            processes.reset.setActualStatus('Powering off the axis');
            // power off the axis
            processes.powerOff.start();
            processes.reset._state := 1;
        1:
            IF processes.powerOff.isIdle() THEN
                // regardless of whether power off worked or not, proceed    
                processes.reset._state := 2;
			END_IF
        2:
            // update the physical axis soft position limit values
            parts.physicalAxis.processes.writeParameter.start(parameterNumber := MC_AxisParameter.SWLimitNeg, value := config.minPositionLimitPhysicalAxis);
            processes.reset._state := 3;
        3:
            IF parts.physicalAxis.processes.writeParameter.isIdle() THEN
                IF parts.physicalAxis.processes.writeParameter.isGood() THEN
                    processes.reset._state := 4;
                ELSE
                    processes.reset.setActualStatus(CONCAT('Could not set the physical SWLimitNeg: ', parts.physicalAxis.processes.writeParameter.actualStatus));
                    processes.reset._state := 999;
				END_IF
			END_IF
        4:
            parts.physicalAxis.processes.writeParameter.start(parameterNumber := MC_AxisParameter.SWLimitPos, value := config.maxPositionLimitPhysicalAxis);
            processes.reset._state := 5;
        5:
            IF parts.physicalAxis.processes.writeParameter.isIdle() THEN
                IF parts.physicalAxis.processes.writeParameter.isGood() THEN
                    processes.reset._state := 6;
                ELSE
                    processes.reset.setActualStatus(CONCAT('Could not set the physical SWLimitPos: ', parts.physicalAxis.processes.writeParameter.actualStatus));
                    processes.reset._state := 999;
				END_IF
			END_IF
        6:
            parts.physicalAxis.processes.writeBoolParameter.start(parameterNumber := MC_AxisParameter.EnableLimitNeg, value := TRUE);
            processes.reset._state := 7;
        7:
            IF parts.physicalAxis.processes.writeBoolParameter.isIdle() THEN
                IF parts.physicalAxis.processes.writeBoolParameter.isGood() THEN
                    processes.reset._state := 8;
                ELSE
                    processes.reset.setActualStatus(CONCAT('Could not set the physical EnableLimitNeg: ', parts.physicalAxis.processes.writeBoolParameter.actualStatus));
                    processes.reset._state := 999;
				END_IF
			END_IF
        8:
            parts.physicalAxis.processes.writeBoolParameter.start(parameterNumber := MC_AxisParameter.EnableLimitPos, value := TRUE);
            processes.reset._state := 9;
        9:
            IF parts.physicalAxis.processes.writeBoolParameter.isIdle() THEN
                IF parts.physicalAxis.processes.writeBoolParameter.isGood() THEN
                    processes.reset._state := 10;
                ELSE
                    processes.reset.setActualStatus(CONCAT('Could not set the physical EnableLimitPos: ', parts.physicalAxis.processes.writeBoolParameter.actualStatus));
                    processes.reset._state := 999;
				END_IF
			END_IF
        10:
            // update the virtual axis soft position limit values
            parts.virtualAxis.processes.writeParameter.start(parameterNumber := MC_AxisParameter.SWLimitNeg, value := config.minPositionLimitVirtualAxis);
            processes.reset._state := 11;
        11:
            IF parts.virtualAxis.processes.writeParameter.isIdle() THEN
                IF parts.virtualAxis.processes.writeParameter.isGood() THEN
                    processes.reset._state := 12;
                ELSE
                    processes.reset.setActualStatus(CONCAT('Could not set the virtual SWLimitNeg: ', parts.virtualAxis.processes.writeParameter.actualStatus));
                    processes.reset._state := 999;
				END_IF
			END_IF
        12:
            parts.virtualAxis.processes.writeParameter.start(parameterNumber := MC_AxisParameter.SWLimitPos, value := config.maxPositionLimitVirtualAxis);
            processes.reset._state := 13;
        13:
            IF parts.virtualAxis.processes.writeParameter.isIdle() THEN
                IF parts.virtualAxis.processes.writeParameter.isGood() THEN
                    processes.reset._state := 14;
                ELSE
                    processes.reset.setActualStatus(CONCAT('Could not set the virtual SWLimitPos: ', parts.virtualAxis.processes.writeParameter.actualStatus));
                    processes.reset._state := 999;
				END_IF
			END_IF
        14:
            parts.virtualAxis.processes.writeBoolParameter.start(parameterNumber := MC_AxisParameter.EnableLimitNeg, value := TRUE);
            processes.reset._state := 15;
        15:
            IF parts.virtualAxis.processes.writeBoolParameter.isIdle() THEN
                IF parts.virtualAxis.processes.writeBoolParameter.isGood() THEN
                    processes.reset._state := 16;
                ELSE
                    processes.reset.setActualStatus(CONCAT('Could not set the virtual EnableLimitNeg: ', parts.virtualAxis.processes.writeBoolParameter.actualStatus));
                    processes.reset._state := 999;
				END_IF
			END_IF
        16:
            parts.virtualAxis.processes.writeBoolParameter.start(parameterNumber := MC_AxisParameter.EnableLimitPos, value := TRUE);
            processes.reset._state := 17;
        17:
            IF parts.virtualAxis.processes.writeBoolParameter.isIdle() THEN
                IF parts.virtualAxis.processes.writeBoolParameter.isGood() THEN
                    processes.reset._state := 18;
                ELSE
                    processes.reset.setActualStatus(CONCAT('Could not set the virtual EnableLimitPos: ', parts.virtualAxis.processes.writeBoolParameter.actualStatus));
                    processes.reset._state := 999;
				END_IF
			END_IF
            
        18:
            // reset the drive channel
            processes.reset.setActualStatus('Resetting the drive channel');
            driveChannel.processes.reset.start();
            processes.reset._state := 19;
        19:
            IF driveChannel.processes.reset.isIdle()  THEN
                IF driveChannel.processes.reset.isGood() THEN
                    processes.reset._state := 20;
                ELSE
                    processes.reset.setActualStatus('Could not reset the drive channels!');
                    processes.reset._state := 999;
                END_IF
            END_IF
            
        20:
            // try to acknowledge the safe state (if present)
            processes.reset.setActualStatus('Resetting safety');
            driveChannel.processes.acknowledgeSafetyError.start();
            processes.reset._state := 21;
        21:
            IF driveChannel.processes.acknowledgeSafetyError.isIdle()  THEN
                IF driveChannel.processes.acknowledgeSafetyError.isGood() THEN
                    processes.reset._state := 22;
                ELSE
                    processes.reset.setActualStatus('Cannot get out of safe state!');
                    processes.reset._state := 999;
                END_IF
            END_IF
        22:
            // reset the drive channel
            processes.reset.setActualStatus('Resetting the drive channel');
            driveChannel.processes.reset.start();
            processes.reset._state := 23;
        23:
            IF driveChannel.processes.reset.isIdle()  THEN
                IF driveChannel.processes.reset.isGood() THEN
                    processes.reset._state := 24;
                ELSE
                    processes.reset.setActualStatus('Could not reset the drive channels!');
                    processes.reset._state := 999;
                END_IF
            END_IF
        24:
            // update the drive channel
            processes.reset.setActualStatus('Updating the drive channel');
            driveChannel.processes.update.start();
            processes.reset._state := 25;
        25:
            IF driveChannel.processes.update.isIdle() AND driveChannel.processes.update.isIdle() THEN
                IF driveChannel.processes.update.isGood() AND driveChannel.processes.update.isGood() THEN
                    processes.reset._state := 26;
                ELSE
                    processes.reset.setActualStatus('Could not update the drive channel!');
                    processes.reset._state := 999;
                END_IF
            END_IF
        26:
            // reset the axis
            processes.reset.setActualStatus('Resetting the axes');
            parts.physicalAxis.processes.reset.start();
            parts.virtualAxis.processes.reset.start();
            processes.reset._state := 27;
        27:
            IF     parts.virtualAxis.processes.reset.isIdle() 
               AND parts.physicalAxis.processes.reset.isIdle()  THEN
                IF     parts.virtualAxis.processes.reset.isGood() 
                   AND parts.physicalAxis.processes.reset.isGood()  THEN
                    processes.reset._state := 1000;
                ELSE
                    processes.reset.setActualStatus('Could not reset the axes');
                    processes.reset._state := 999;
                END_IF
            END_IF
        999:
            // error!
            processes.reset.setBad();
            processes.reset.setFinished();
        1000:
            processes.reset.setActualStatus('Reset');
            // ok done
            processes.reset.setFinished();
            processes.reset.setGood();
    END_CASE
    
END_IF
END_METHOD

METHOD callOnce : BOOL
VAR_INPUT
    dcTime : LINT; 
	targetPosDeg  : LREAL; // degrees
	targetVeloDegPerSec : LREAL; // degrees/sec
	targetAccDegPerSec2  : LREAL; // degrees/sec2
    trackingStart : LREAL; // degrees
    modelDelta : LREAL; // degrees
END_VAR
VAR_IN_OUT
    isTracking : BOOL;
END_VAR
// run the setpoint generators
_setGen( 
    dcTime                      := dcTime,
    tracking                    := isTracking,
    virtual                     := parts.virtualAxis.axis_ref, 
    physical                    := parts.physicalAxis.axis_ref, 
    targetPos                   := targetPosDeg, 
    targetVelo                  := targetVeloDegPerSec, 
    targetAcc                   := targetAccDegPerSec2, 
    trackingStart               := trackingStart,
    velocityLimit               := config.velocityLimit,
    accelerationLimit           := config.accelerationLimit,
    minTrackingPositionSetpoint := config.minPositionSetpoint,
    maxTrackingPositionSetpoint := config.maxPositionSetpoint,
    minVirtualPositionSetpoint  := config.minPositionLimitVirtualAxis,
    maxVirtualPositionSetpoint  := config.maxPositionLimitVirtualAxis,
    limitReached                => setPosLimitReached);


// apply the position correction
IF parts.physicalAxis.axis_ref.Status.Homed THEN
    parts.physicalAxis.setPositionCorrection(lidaAveragePosition.degrees.value - parts.physicalAxis.axis_ref.NcToPlc.ActPosWithoutPosCorrection);
ELSE
    parts.physicalAxis.setPositionCorrection(0.0);
END_IF


// calculate the average and RMS deviation
_deviationCalculator(in := parts.physicalAxis.axis_ref.NcToPlc.ActPos - parts.physicalAxis.axis_ref.NcToPlc.SetPos );
deviation1SecAverage(newDegreesValue := _deviationCalculator.avg);
deviation1SecRMS(newDegreesValue := _deviationCalculator.rms);

// keep a local copy of the isTracking variable
_isTracking := isTracking;
END_METHOD

METHOD _moveAbsolute
VAR_INPUT
END_VAR
VAR
    positionDegrees : LREAL;
END_VAR
IF processes.moveAbsolute.isBusy() THEN
    
    IF NOT processes.moveAbsolute.isStarted() THEN
        
        targetStart(newDegreesValue := AxesMoveUnitsToDeg(units := processes.moveAbsolute.get.units, value := processes.moveAbsolute.get.value));
        
        parts.virtualAxis.processes.moveAbsolute.start(position := targetStart.degrees.value + processes.moveAbsolute.get.offset, maxVelocity := config.maxVelocitySetpoint);

        processes.moveAbsolute.setStarted();
            
	END_IF

    // update the statuses
    processes.moveAbsolute.statuses.busyStatus(isBusy := parts.virtualAxis.processes.moveAbsolute.statuses.busyStatus.isBusy);
    processes.moveAbsolute.statuses.healthStatus(
        isGood := parts.virtualAxis.processes.moveAbsolute.statuses.healthStatus.isGood,
        hasWarning := parts.virtualAxis.processes.moveAbsolute.statuses.healthStatus.hasWarning);
    processes.moveAbsolute.setActualStatus(parts.virtualAxis.processes.moveAbsolute.actualStatus);

END_IF
END_METHOD

METHOD _moveRelative
VAR_INPUT
END_VAR
VAR
    distanceDegrees : LREAL;
END_VAR
IF processes.moveRelative.isBusy() THEN
    
    IF NOT processes.moveRelative.isStarted() THEN
        
        distanceDegrees := AxesMoveUnitsToDeg(units := processes.moveRelative.get.units, value := processes.moveRelative.get.value);
        
        parts.virtualAxis.processes.moveRelative.start(distance := distanceDegrees, maxVelocity := config.maxVelocitySetpoint);
    
        processes.moveRelative.setStarted();
            
	END_IF

    // update the statuses
    processes.moveRelative.statuses.busyStatus(isBusy := parts.virtualAxis.processes.moveRelative.statuses.busyStatus.isBusy);
    processes.moveRelative.statuses.healthStatus(
        isGood := parts.virtualAxis.processes.moveRelative.statuses.healthStatus.isGood,
        hasWarning := parts.virtualAxis.processes.moveRelative.statuses.healthStatus.hasWarning);
    processes.moveRelative.setActualStatus(parts.virtualAxis.processes.moveRelative.actualStatus);

END_IF
END_METHOD

END_FUNCTION_BLOCK

// ---- MTCS/Axes/StateMachines/AxesRotationAxis.TcPOU
FUNCTION_BLOCK AxesRotationAxis EXTENDS SM_AxesRotationAxis
VAR_INPUT
END_VAR
VAR_OUTPUT
END_VAR
VAR 
    // setpoint generator
	{attribute 'OPC.UA.DA' := '0'}
    _setGen : AxesExternalSetpointGenerator;
    
    // helpers
	{attribute 'OPC.UA.DA' := '0'}
    _powerOnHelper : AxesPowerOnHelper;
	{attribute 'OPC.UA.DA' := '0'}
    _powerOffHelper : AxesPowerOffHelper;
	{attribute 'OPC.UA.DA' := '0'}
    _homingHelper : AxesHomingHelper;
	{attribute 'OPC.UA.DA' := '0'}
    _moveOutOfLimitSwitchHelper : AxesMoveOutOfLimitSwitchHelper;
	{attribute 'OPC.UA.DA' := '0'}
    _stopHelper : AxesStopHelper;
	{attribute 'OPC.UA.DA' := '0'}
    _quickStopHelper : AxesQuickStopHelper;
	{attribute 'OPC.UA.DA' := '0'}
    _setPositionHelper : AxesSetPositionHelper;
    
    // RMS and average setpoint deviation calculator
	{attribute 'OPC.UA.DA' := '0'}
    _deviationCalculator: AverageAndRmsCalculator;
    // local copy of the isTracking flag
	{attribute 'OPC.UA.DA' := '0'}
    _isTracking: BOOL;
	{attribute 'OPC.UA.DA' := '0'}
    _moveRelativeCalculator : AxesMoveRelativeCalculator;
	{attribute 'OPC.UA.DA' := '0'}
    _moveAbsoluteCalculator : AxesMoveAbsoluteCalculator;
    
END_VAR

_update();

_resetting();


_powerOnHelper(
    id                      := id,
    setpointGenerator       := _setGen,
    powerOn                 := processes.powerOn,
    stop                    := processes.stop,
    reset                   := processes.reset,
    virtual                 := parts.virtualAxis,
    physical                := parts.physicalAxis,
    targetStart             := targetStart,
    pAblAxis                := 0,
    pAblDriveChannel        := 0,
    pAblSetpointGenerator   := 0);
    
_powerOffHelper(
    setpointGenerator       := _setGen,
    powerOff                := processes.powerOff,
    stop                    := processes.stop,
    virtual                 := parts.virtualAxis,
    physical                := parts.physicalAxis,
    pAblAxis                := 0,
    pAblDriveChannel        := 0,
    pAblSetpointGenerator   := 0);


_moveOutOfLimitSwitchHelper(
    setpointGenerator               := _setGen,
    positiveLimitSwitchError        := positiveLimitSwitchError,
    negativeLimitSwitchError        := negativeLimitSwitchError,
    positiveLimitSwitchInput        := config.positiveLimitSwitchInput,
    negativeLimitSwitchInput        := config.negativeLimitSwitchInput,
    moveOutOfLimitSwitchDistance    := config.moveOutOfLimitSwitchDistance,
    moveOutOfLimitSwitch            := processes.moveOutOfLimitSwitch,
    moveRelative                    := processes.moveRelative,
    powerOn                         := processes.powerOn,
    reset                           := processes.reset,
    virtual                         := parts.virtualAxis,
    physical                        := parts.physicalAxis,
    driveChannel                    := mainDriveChannel);

_moveAbsolute();
_moveRelative();
_moveVelocity();

_stopHelper(
    setpointGenerator   := _setGen,
    stop                := processes.stop,
    virtual             := parts.virtualAxis,
    physical            := parts.physicalAxis);
    
_quickStopHelper(
    deceleration        := config.quickStopDeceleration, 
    jerk                := config.quickStopJerk,
    setpointGenerator   := _setGen,
    quickStop           := processes.quickStop,
    virtual             := parts.virtualAxis,
    physical            := parts.physicalAxis);
    
_setPositionHelper(
    setpointGenerator   := _setGen,
    setPosition         := processes.setPosition,
    virtual             := parts.virtualAxis,
    physical            := parts.physicalAxis);


_update();

METHOD callOnce : BOOL
VAR_INPUT
    dcTime : LINT; 
	targetPosDeg  : LREAL; // degrees
	targetVeloDegPerSec : LREAL; // degrees/sec
	targetAccDegPerSec2  : LREAL; // degrees/sec2
    trackingStart : LREAL; // degrees
END_VAR
VAR_IN_OUT
    isTracking : BOOL;
END_VAR
// run the setpoint generators
_setGen( 
    dcTime                      := dcTime,
    tracking                    := isTracking,
    virtual                     := parts.virtualAxis.axis_ref, 
    physical                    := parts.physicalAxis.axis_ref, 
    targetPos                   := targetPosDeg, 
    targetVelo                  := targetVeloDegPerSec, 
    targetAcc                   := targetAccDegPerSec2, 
    trackingStart               := trackingStart,
    velocityLimit               := config.velocityLimit,
    accelerationLimit           := config.accelerationLimit,
    minTrackingPositionSetpoint := config.minPositionSetpoint,
    maxTrackingPositionSetpoint := config.maxPositionSetpoint,
    minVirtualPositionSetpoint  := config.minPositionLimitVirtualAxis,
    maxVirtualPositionSetpoint  := config.maxPositionLimitVirtualAxis,
    limitReached                => setPosLimitReached);

// calculate the average and RMS deviation
_deviationCalculator(in := parts.physicalAxis.axis_ref.NcToPlc.ActPos - parts.physicalAxis.axis_ref.NcToPlc.SetPos );
deviation1SecAverage(newDegreesValue := _deviationCalculator.avg);
deviation1SecRMS(newDegreesValue := _deviationCalculator.rms);

// keep a local copy of the isTracking variable
_isTracking := isTracking;
END_METHOD

METHOD _moveVelocity
VAR_INPUT
END_VAR
VAR
    velocityDegPerSec : LREAL;
END_VAR
IF processes.moveVelocity.isBusy() THEN
    
    IF NOT processes.moveVelocity.isStarted() THEN
        
        velocityDegPerSec := AxesMoveVelocityUnitsToDegPerSec(units := processes.moveVelocity.get.units, value := processes.moveVelocity.get.value);
        
        parts.virtualAxis.processes.moveVelocity.start(value := velocityDegPerSec);
    
        processes.moveVelocity.setStarted();
            
	END_IF

    // update the statuses
    processes.moveVelocity.statuses.busyStatus(isBusy := parts.virtualAxis.processes.moveVelocity.statuses.busyStatus.isBusy);
    processes.moveVelocity.statuses.healthStatus(
        isGood := parts.virtualAxis.processes.moveVelocity.statuses.healthStatus.isGood,
        hasWarning := parts.virtualAxis.processes.moveVelocity.statuses.healthStatus.hasWarning);
    processes.moveVelocity.setActualStatus(parts.virtualAxis.processes.moveVelocity.actualStatus);

END_IF
END_METHOD

METHOD _update : LREAL
VAR_INPUT
END_VAR
VAR
END_VAR
// update the superclass
SUPER^(
    config := config,
    driveChannel := driveChannel,
    mainDriveChannel := mainDriveChannel);
    
// update the limit switches
positiveLimitSwitchError := NOT GETBIT32(inVal32 := INT_TO_DWORD(driveChannel.digitalInputs), bitNo := config.positiveLimitSwitchInput);
negativeLimitSwitchError := NOT GETBIT32(inVal32 := INT_TO_DWORD(driveChannel.digitalInputs), bitNo := config.negativeLimitSwitchInput);

// update the actual position/velocity/acceleration
actPos(newDegreesValue := parts.physicalAxis.axis_ref.NcToPlc.ActPos);
actVelo(newDegreesPerSecondValue := parts.physicalAxis.axis_ref.NcToPlc.ActVelo);
actAcc(newDegreesPerSquareSecondValue := parts.physicalAxis.axis_ref.NcToPlc.ActAcc);
setPos(newDegreesValue := parts.physicalAxis.axis_ref.NcToPlc.SetPos);
setVelo(newDegreesPerSecondValue := parts.physicalAxis.axis_ref.NcToPlc.SetVelo);
setAcc(newDegreesPerSquareSecondValue := parts.physicalAxis.axis_ref.NcToPlc.SetAcc);
IF parts.physicalAxis.axis_ref.Status.ExtSetPointGenEnabled THEN
    targetPos(newDegreesValue := parts.physicalAxis.axis_ref.PlcToNc.ExtSetPos);
    targetOffset(newDegreesValue := parts.virtualAxis.actPos.degrees.value - targetStart.degrees.value);
ELSE
    targetPos(newDegreesValue := parts.physicalAxis.axis_ref.NcToPlc.TargetPos);
    targetOffset(newDegreesValue := 0.0);
END_IF

// update the actual torque feedback on the telescope side
actTorque(newNewtonmeterValue := driveChannel.actualTorqueFeedback.newtonmeter.value * 1440);
END_METHOD

METHOD _moveRelative
VAR_INPUT
END_VAR
VAR
    distanceDegrees : LREAL;
END_VAR
IF processes.moveRelative.isBusy() THEN
    
    IF NOT processes.moveRelative.isStarted() THEN
        
        distanceDegrees := AxesMoveUnitsToDeg(units := processes.moveRelative.get.units, value := processes.moveRelative.get.value);
        
        parts.virtualAxis.processes.moveRelative.start(distance := distanceDegrees, maxVelocity := config.maxVelocitySetpoint);
    
        processes.moveRelative.setStarted();
    ELSE
        
        // update the statuses
        processes.moveRelative.statuses.healthStatus(
            isGood := parts.virtualAxis.processes.moveRelative.statuses.healthStatus.isGood,
            hasWarning := parts.virtualAxis.processes.moveRelative.statuses.healthStatus.hasWarning);
        processes.moveRelative.setActualStatus(parts.virtualAxis.processes.moveRelative.actualStatus);
        processes.moveRelative.statuses.busyStatus(isBusy := parts.virtualAxis.processes.moveRelative.statuses.busyStatus.isBusy);
    
	END_IF
END_IF
(*IF processes.moveRelative.isBusy() THEN
    
    IF NOT processes.moveRelative.isStarted() THEN
        
        distanceDegrees := AxesMoveUnitsToDeg(units := processes.moveRelative.get.units, value := processes.moveRelative.get.value);
        
        _moveRelativeCalculator(
            distance     := distanceDegrees, 
            trackingVelo := _setGen.targetVelo,
            minPos       := config.minPositionLimitVirtualAxis,
            maxPos       := config.maxPositionLimitVirtualAxis,
            actPos       := actPos.degrees.value,
            doMostTravel := processes.moveRelative.get.preferMostTravel);
        
        IF _moveRelativeCalculator.outOfRange THEN
            processes.moveRelative.setFinished();
            processes.moveRelative.setActualStatus('Out of limits!');
            processes.moveRelative.setBad();
        ELSE
            parts.virtualAxis.processes.moveRelative.start(distance := _moveRelativeCalculator.adjustedDistance, maxVelocity := config.maxVelocitySetpoint);
            processes.moveRelative.setStarted();
        END_IF
        
    ELSE
        // update the statuses
        processes.moveRelative.statuses.busyStatus(isBusy := parts.virtualAxis.processes.moveRelative.statuses.busyStatus.isBusy);
        processes.moveRelative.statuses.healthStatus(
            isGood := parts.virtualAxis.processes.moveRelative.statuses.healthStatus.isGood,
            hasWarning := parts.virtualAxis.processes.moveRelative.statuses.healthStatus.hasWarning);
        processes.moveRelative.setActualStatus(parts.virtualAxis.processes.moveRelative.actualStatus);

	END_IF

END_IF*)
END_METHOD

METHOD _moveAbsolute
VAR_INPUT
END_VAR
VAR
    positionDegrees : LREAL;
END_VAR
IF processes.moveAbsolute.isBusy() THEN
    
    IF NOT processes.moveAbsolute.isStarted() THEN
        
        targetStart(newDegreesValue := AxesMoveUnitsToDeg(units := processes.moveAbsolute.get.units, value := processes.moveAbsolute.get.value));
        
        parts.virtualAxis.processes.moveAbsolute.start(position := targetStart.degrees.value + processes.moveAbsolute.get.offset, maxVelocity := config.maxVelocitySetpoint);

        processes.moveAbsolute.setStarted();
        
    END_IF

    IF parts.virtualAxis.processes.moveAbsolute.isIdle() THEN
        
        IF parts.virtualAxis.processes.moveAbsolute.isGood() THEN
            processes.moveAbsolute.setGood();
        ELSE
            processes.moveAbsolute.setBad();
		END_IF
        
        processes.moveAbsolute.setActualStatus(parts.virtualAxis.processes.moveAbsolute.actualStatus);
        processes.moveAbsolute.setFinished();
    
	END_IF
    
END_IF
(*IF processes.moveAbsolute.isBusy() THEN
    
    IF NOT processes.moveAbsolute.isStarted() THEN
        
        _moveAbsoluteCalculator(
            targetPos := AxesMoveUnitsToDeg(units := processes.moveAbsolute.get.units, value := processes.moveAbsolute.get.value),
            trackingVelo := _setGen.targetVelo,
            minPos := config.minPositionLimitVirtualAxis,
            maxPos := config.maxPositionLimitVirtualAxis,
            actPos := parts.virtualAxis.actPos.degrees.value,
            doMostTravel := FALSE); // get there the quickest possible
        
        IF _moveAbsoluteCalculator.outOfRange THEN
            processes.moveAbsolute.setActualStatus('Out of limits!');
            processes.moveAbsolute.setBad();
            processes.moveAbsolute.setFinished();
        ELSE
            targetStart(newDegreesValue := _moveAbsoluteCalculator.adjustedPos);
            parts.virtualAxis.processes.moveAbsolute.start(position := targetStart.degrees.value, maxVelocity := config.maxVelocitySetpoint);
            processes.moveAbsolute.setStarted();
		END_IF
            
    ELSE
        // update the statuses
        processes.moveAbsolute.statuses.busyStatus(isBusy := parts.virtualAxis.processes.moveAbsolute.statuses.busyStatus.isBusy);
        processes.moveAbsolute.statuses.healthStatus(
            isGood := parts.virtualAxis.processes.moveAbsolute.statuses.healthStatus.isGood,
            hasWarning := parts.virtualAxis.processes.moveAbsolute.statuses.healthStatus.hasWarning);
        processes.moveAbsolute.setActualStatus(parts.virtualAxis.processes.moveAbsolute.actualStatus);

	END_IF

END_IF*)
END_METHOD

METHOD _resetting : LREAL
VAR_INPUT
END_VAR
IF processes.reset.isBusy() THEN
    
    IF NOT processes.reset.isStarted() THEN
        processes.reset._state := 0;
        processes.reset.setStarted();
	END_IF
    
    CASE processes.reset._state OF
        0:
            // reset all processes so that they are green again
            processes.moveAbsolute.resetIfIdle();
            processes.moveOutOfLimitSwitch.resetIfIdle();
            processes.moveRelative.resetIfIdle();
            processes.moveVelocity.resetIfIdle();
            processes.powerOff.resetIfIdle();
            processes.powerOn.resetIfIdle();
            processes.quickStop.resetIfIdle();
            processes.setPosition.resetIfIdle();
            processes.stop.resetIfIdle();
            
            processes.reset.setActualStatus('Powering off the axis');
            // power off the axis
            processes.powerOff.start();
            processes.reset._state := 1;
        1:
            IF processes.powerOff.isIdle() THEN
                // regardless of whether power off worked or not, proceed    
                processes.reset._state := 2;
			END_IF
        2:
            // update the physical axis soft position limit values
            parts.physicalAxis.processes.writeParameter.start(parameterNumber := MC_AxisParameter.AxisEncoderOffset, value := config.motorEncoderOffset);
            processes.reset._state := 3;
        3:
            IF parts.physicalAxis.processes.writeParameter.isIdle() THEN
                IF parts.physicalAxis.processes.writeParameter.isGood() THEN
                    processes.reset._state := 4;
                ELSE
                    processes.reset.setActualStatus(CONCAT('Could not set the motor encoder offset: ', parts.physicalAxis.processes.writeParameter.actualStatus));
                    processes.reset._state := 999;
				END_IF
			END_IF
        4:
            // update the physical axis soft position limit values
            parts.physicalAxis.processes.writeParameter.start(parameterNumber := MC_AxisParameter.SWLimitNeg, value := config.minPositionLimitPhysicalAxis);
            processes.reset._state := 5;
        5:
            IF parts.physicalAxis.processes.writeParameter.isIdle() THEN
                IF parts.physicalAxis.processes.writeParameter.isGood() THEN
                    processes.reset._state := 6;
                ELSE
                    processes.reset.setActualStatus(CONCAT('Could not set the physical SWLimitNeg: ', parts.physicalAxis.processes.writeParameter.actualStatus));
                    processes.reset._state := 999;
				END_IF
			END_IF
        6:
            parts.physicalAxis.processes.writeParameter.start(parameterNumber := MC_AxisParameter.SWLimitPos, value := config.maxPositionLimitPhysicalAxis);
            processes.reset._state := 7;
        7:
            IF parts.physicalAxis.processes.writeParameter.isIdle() THEN
                IF parts.physicalAxis.processes.writeParameter.isGood() THEN
                    processes.reset._state := 8;
                ELSE
                    processes.reset.setActualStatus(CONCAT('Could not set the physical SWLimitPos: ', parts.physicalAxis.processes.writeParameter.actualStatus));
                    processes.reset._state := 999;
				END_IF
			END_IF
        8:
            parts.physicalAxis.processes.writeBoolParameter.start(parameterNumber := MC_AxisParameter.EnableLimitNeg, value := TRUE);
            processes.reset._state := 9;
        9:
            IF parts.physicalAxis.processes.writeBoolParameter.isIdle() THEN
                IF parts.physicalAxis.processes.writeBoolParameter.isGood() THEN
                    processes.reset._state := 10;
                ELSE
                    processes.reset.setActualStatus(CONCAT('Could not set the physical EnableLimitNeg: ', parts.physicalAxis.processes.writeBoolParameter.actualStatus));
                    processes.reset._state := 999;
				END_IF
			END_IF
        10:
            parts.physicalAxis.processes.writeBoolParameter.start(parameterNumber := MC_AxisParameter.EnableLimitPos, value := TRUE);
            processes.reset._state := 11;
        11:
            IF parts.physicalAxis.processes.writeBoolParameter.isIdle() THEN
                IF parts.physicalAxis.processes.writeBoolParameter.isGood() THEN
                    processes.reset._state := 12;
                ELSE
                    processes.reset.setActualStatus(CONCAT('Could not set the physical EnableLimitPos: ', parts.physicalAxis.processes.writeBoolParameter.actualStatus));
                    processes.reset._state := 999;
				END_IF
			END_IF
        12:
            // update the virtual axis soft position limit values
            parts.virtualAxis.processes.writeParameter.start(parameterNumber := MC_AxisParameter.SWLimitNeg, value := config.minPositionLimitVirtualAxis);
            processes.reset._state := 13;
        13:
            IF parts.virtualAxis.processes.writeParameter.isIdle() THEN
                IF parts.virtualAxis.processes.writeParameter.isGood() THEN
                    processes.reset._state := 14;
                ELSE
                    processes.reset.setActualStatus(CONCAT('Could not set the virtual SWLimitNeg: ', parts.virtualAxis.processes.writeParameter.actualStatus));
                    processes.reset._state := 999;
				END_IF
			END_IF
        14:
            parts.virtualAxis.processes.writeParameter.start(parameterNumber := MC_AxisParameter.SWLimitPos, value := config.maxPositionLimitVirtualAxis);
            processes.reset._state := 15;
        15:
            IF parts.virtualAxis.processes.writeParameter.isIdle() THEN
                IF parts.virtualAxis.processes.writeParameter.isGood() THEN
                    processes.reset._state := 16;
                ELSE
                    processes.reset.setActualStatus(CONCAT('Could not set the virtual SWLimitPos: ', parts.virtualAxis.processes.writeParameter.actualStatus));
                    processes.reset._state := 999;
				END_IF
			END_IF
        16:
            parts.virtualAxis.processes.writeBoolParameter.start(parameterNumber := MC_AxisParameter.EnableLimitNeg, value := TRUE);
            processes.reset._state := 17;
        17:
            IF parts.virtualAxis.processes.writeBoolParameter.isIdle() THEN
                IF parts.virtualAxis.processes.writeBoolParameter.isGood() THEN
                    processes.reset._state := 18;
                ELSE
                    processes.reset.setActualStatus(CONCAT('Could not set the virtual EnableLimitNeg: ', parts.virtualAxis.processes.writeBoolParameter.actualStatus));
                    processes.reset._state := 999;
				END_IF
			END_IF
        18:
            parts.virtualAxis.processes.writeBoolParameter.start(parameterNumber := MC_AxisParameter.EnableLimitPos, value := TRUE);
            processes.reset._state := 19;
        19:
            IF parts.virtualAxis.processes.writeBoolParameter.isIdle() THEN
                IF parts.virtualAxis.processes.writeBoolParameter.isGood() THEN
                    processes.reset._state := 20;
                ELSE
                    processes.reset.setActualStatus(CONCAT('Could not set the virtual EnableLimitPos: ', parts.virtualAxis.processes.writeBoolParameter.actualStatus));
                    processes.reset._state := 999;
				END_IF
			END_IF
            
        20:
            // try to acknowledge the safe state (if present)
            processes.reset.setActualStatus('Resetting safety');
            driveChannel.processes.acknowledgeSafetyError.start();
            processes.reset._state := 21;
        21:
            IF driveChannel.processes.acknowledgeSafetyError.isIdle()  THEN
                IF driveChannel.processes.acknowledgeSafetyError.isGood() THEN
                    processes.reset._state := 22;
                ELSE
                    processes.reset.setActualStatus('Cannot get out of safe state!');
                    processes.reset._state := 999;
                END_IF
            END_IF
        22:
            // reset the drive channel
            processes.reset.setActualStatus('Resetting the drive channel');
            driveChannel.processes.reset.start();
            processes.reset._state := 23;
        23:
            IF driveChannel.processes.reset.isIdle()  THEN
                IF driveChannel.processes.reset.isGood() THEN
                    processes.reset._state := 24;
                ELSE
                    processes.reset.setActualStatus('Could not reset the drive channels!');
                    processes.reset._state := 999;
                END_IF
            END_IF
        24:
            // update the drive channel
            processes.reset.setActualStatus('Updating the drive channel');
            driveChannel.processes.update.start();
            processes.reset._state := 25;
        25:
            IF driveChannel.processes.update.isIdle() AND driveChannel.processes.update.isIdle() THEN
                IF driveChannel.processes.update.isGood() AND driveChannel.processes.update.isGood() THEN
                    processes.reset._state := 26;
                ELSE
                    processes.reset.setActualStatus('Could not update the drive channel!');
                    processes.reset._state := 999;
                END_IF
            END_IF
        26:
            // reset the axis
            processes.reset.setActualStatus('Resetting the axes');
            parts.physicalAxis.processes.reset.start();
            parts.virtualAxis.processes.reset.start();
            processes.reset._state := 27;
        27:
            IF     parts.virtualAxis.processes.reset.isIdle() 
               AND parts.physicalAxis.processes.reset.isIdle()  THEN
                IF     parts.virtualAxis.processes.reset.isGood() 
                   AND parts.physicalAxis.processes.reset.isGood()  THEN
                    processes.reset._state := 1000;
                ELSE
                    processes.reset.setActualStatus('Could not reset the axes');
                    processes.reset._state := 999;
                END_IF
            END_IF
        999:
            // error!
            processes.reset.setBad();
            processes.reset.setFinished();
        1000:
            processes.reset.setActualStatus('Reset');
            // ok done
            processes.reset.setFinished();
            processes.reset.setGood();
    END_CASE
    
END_IF
END_METHOD

END_FUNCTION_BLOCK

// ---- MTCS/Axes/StateMachines/AxesIO.TcPOU
FUNCTION_BLOCK AxesIO EXTENDS SM_AxesIO
VAR_INPUT
END_VAR
VAR_OUTPUT
END_VAR
VAR
    _testVar : BOOL; // without any variable, the superclass attributes are not visible in the UA address space
END_VAR

SUPER^();

// do stuff

//SUPER^();

END_FUNCTION_BLOCK

// ---- MTCS/Axes/StateMachines/AxesPointingModelsSetup.TcPOU
FUNCTION_BLOCK AxesPointingModelsSetup EXTENDS SM_AxesPointingModelsSetup
VAR_INPUT
END_VAR
VAR_OUTPUT
END_VAR
VAR
	{attribute 'OPC.UA.DA' := '0'}
    _onFirstStartCurrentAction : INT;
END_VAR

SUPER^();

_onFirstStart();

METHOD FB_init : BOOL
VAR_INPUT
	bInitRetains : BOOL; // if TRUE, the retain variables are initialized (warm start / cold start)
	bInCopyCode : BOOL;  // if TRUE, the instance afterwards gets moved into the copy code (online change)
END_VAR
parts.model0.parts.configManager.configure(
    editableConfigAddress       := ADR(parts.model0.editableConfig),
    activeConfigAddress         := ADR(parts.model0.config),
    configLength                := SIZEOF(parts.model0.editableConfig),
    editableConfigSymbolName    := CONCAT(CONCAT(GLOBAL.config.AXES_TPOINT_EDITABLE_CONFIG_SYMBOL_PREFIX, 'model0'), GLOBAL.config.AXES_TPOINT_EDITABLE_CONFIG_SYMBOL_SUFFIX),
    activeConfigSymbolName      := CONCAT(CONCAT(GLOBAL.config.AXES_TPOINT_ACTIVE_CONFIG_SYMBOL_PREFIX, 'model0'), GLOBAL.config.AXES_TPOINT_ACTIVE_CONFIG_SYMBOL_SUFFIX),
    configFilePath              := CONCAT(CONCAT(GLOBAL.config.AXES_TPOINT_CONFIG_FILE_PATH_PREFIX, 'model0'), GLOBAL.config.AXES_TPOINT_CONFIG_FILE_PATH_SUFFIX));
    
parts.model1.parts.configManager.configure(
    editableConfigAddress       := ADR(parts.model1.editableConfig),
    activeConfigAddress         := ADR(parts.model1.config),
    configLength                := SIZEOF(parts.model1.editableConfig),
    editableConfigSymbolName    := CONCAT(CONCAT(GLOBAL.config.AXES_TPOINT_EDITABLE_CONFIG_SYMBOL_PREFIX, 'model1'), GLOBAL.config.AXES_TPOINT_EDITABLE_CONFIG_SYMBOL_SUFFIX),
    activeConfigSymbolName      := CONCAT(CONCAT(GLOBAL.config.AXES_TPOINT_ACTIVE_CONFIG_SYMBOL_PREFIX, 'model1'), GLOBAL.config.AXES_TPOINT_ACTIVE_CONFIG_SYMBOL_SUFFIX),
    configFilePath              := CONCAT(CONCAT(GLOBAL.config.AXES_TPOINT_CONFIG_FILE_PATH_PREFIX, 'model1'), GLOBAL.config.AXES_TPOINT_CONFIG_FILE_PATH_SUFFIX));
    
parts.model2.parts.configManager.configure(
    editableConfigAddress       := ADR(parts.model2.editableConfig),
    activeConfigAddress         := ADR(parts.model2.config),
    configLength                := SIZEOF(parts.model2.editableConfig),
    editableConfigSymbolName    := CONCAT(CONCAT(GLOBAL.config.AXES_TPOINT_EDITABLE_CONFIG_SYMBOL_PREFIX, 'model2'), GLOBAL.config.AXES_TPOINT_EDITABLE_CONFIG_SYMBOL_SUFFIX),
    activeConfigSymbolName      := CONCAT(CONCAT(GLOBAL.config.AXES_TPOINT_ACTIVE_CONFIG_SYMBOL_PREFIX, 'model2'), GLOBAL.config.AXES_TPOINT_ACTIVE_CONFIG_SYMBOL_SUFFIX),
    configFilePath              := CONCAT(CONCAT(GLOBAL.config.AXES_TPOINT_CONFIG_FILE_PATH_PREFIX, 'model2'), GLOBAL.config.AXES_TPOINT_CONFIG_FILE_PATH_SUFFIX));
parts.model3.parts.configManager.configure(
    editableConfigAddress       := ADR(parts.model3.editableConfig),
    activeConfigAddress         := ADR(parts.model3.config),
    configLength                := SIZEOF(parts.model3.editableConfig),
    editableConfigSymbolName    := CONCAT(CONCAT(GLOBAL.config.AXES_TPOINT_EDITABLE_CONFIG_SYMBOL_PREFIX, 'model3'), GLOBAL.config.AXES_TPOINT_EDITABLE_CONFIG_SYMBOL_SUFFIX),
    activeConfigSymbolName      := CONCAT(CONCAT(GLOBAL.config.AXES_TPOINT_ACTIVE_CONFIG_SYMBOL_PREFIX, 'model3'), GLOBAL.config.AXES_TPOINT_ACTIVE_CONFIG_SYMBOL_SUFFIX),
    configFilePath              := CONCAT(CONCAT(GLOBAL.config.AXES_TPOINT_CONFIG_FILE_PATH_PREFIX, 'model3'), GLOBAL.config.AXES_TPOINT_CONFIG_FILE_PATH_SUFFIX));
parts.model4.parts.configManager.configure(
    editableConfigAddress       := ADR(parts.model4.editableConfig),
    activeConfigAddress         := ADR(parts.model4.config),
    configLength                := SIZEOF(parts.model4.editableConfig),
    editableConfigSymbolName    := CONCAT(CONCAT(GLOBAL.config.AXES_TPOINT_EDITABLE_CONFIG_SYMBOL_PREFIX, 'model4'), GLOBAL.config.AXES_TPOINT_EDITABLE_CONFIG_SYMBOL_SUFFIX),
    activeConfigSymbolName      := CONCAT(CONCAT(GLOBAL.config.AXES_TPOINT_ACTIVE_CONFIG_SYMBOL_PREFIX, 'model4'), GLOBAL.config.AXES_TPOINT_ACTIVE_CONFIG_SYMBOL_SUFFIX),
    configFilePath              := CONCAT(CONCAT(GLOBAL.config.AXES_TPOINT_CONFIG_FILE_PATH_PREFIX, 'model4'), GLOBAL.config.AXES_TPOINT_CONFIG_FILE_PATH_SUFFIX));
parts.model5.parts.configManager.configure(
    editableConfigAddress       := ADR(parts.model5.editableConfig),
    activeConfigAddress         := ADR(parts.model5.config),
    configLength                := SIZEOF(parts.model5.editableConfig),
    editableConfigSymbolName    := CONCAT(CONCAT(GLOBAL.config.AXES_TPOINT_EDITABLE_CONFIG_SYMBOL_PREFIX, 'model5'), GLOBAL.config.AXES_TPOINT_EDITABLE_CONFIG_SYMBOL_SUFFIX),
    activeConfigSymbolName      := CONCAT(CONCAT(GLOBAL.config.AXES_TPOINT_ACTIVE_CONFIG_SYMBOL_PREFIX, 'model5'), GLOBAL.config.AXES_TPOINT_ACTIVE_CONFIG_SYMBOL_SUFFIX),
    configFilePath              := CONCAT(CONCAT(GLOBAL.config.AXES_TPOINT_CONFIG_FILE_PATH_PREFIX, 'model5'), GLOBAL.config.AXES_TPOINT_CONFIG_FILE_PATH_SUFFIX));
parts.model6.parts.configManager.configure(
    editableConfigAddress       := ADR(parts.model6.editableConfig),
    activeConfigAddress         := ADR(parts.model6.config),
    configLength                := SIZEOF(parts.model6.editableConfig),
    editableConfigSymbolName    := CONCAT(CONCAT(GLOBAL.config.AXES_TPOINT_EDITABLE_CONFIG_SYMBOL_PREFIX, 'model6'), GLOBAL.config.AXES_TPOINT_EDITABLE_CONFIG_SYMBOL_SUFFIX),
    activeConfigSymbolName      := CONCAT(CONCAT(GLOBAL.config.AXES_TPOINT_ACTIVE_CONFIG_SYMBOL_PREFIX, 'model6'), GLOBAL.config.AXES_TPOINT_ACTIVE_CONFIG_SYMBOL_SUFFIX),
    configFilePath              := CONCAT(CONCAT(GLOBAL.config.AXES_TPOINT_CONFIG_FILE_PATH_PREFIX, 'model6'), GLOBAL.config.AXES_TPOINT_CONFIG_FILE_PATH_SUFFIX));
parts.model7.parts.configManager.configure(
    editableConfigAddress       := ADR(parts.model7.editableConfig),
    activeConfigAddress         := ADR(parts.model7.config),
    configLength                := SIZEOF(parts.model7.editableConfig),
    editableConfigSymbolName    := CONCAT(CONCAT(GLOBAL.config.AXES_TPOINT_EDITABLE_CONFIG_SYMBOL_PREFIX, 'model7'), GLOBAL.config.AXES_TPOINT_EDITABLE_CONFIG_SYMBOL_SUFFIX),
    activeConfigSymbolName      := CONCAT(CONCAT(GLOBAL.config.AXES_TPOINT_ACTIVE_CONFIG_SYMBOL_PREFIX, 'model7'), GLOBAL.config.AXES_TPOINT_ACTIVE_CONFIG_SYMBOL_SUFFIX),
    configFilePath              := CONCAT(CONCAT(GLOBAL.config.AXES_TPOINT_CONFIG_FILE_PATH_PREFIX, 'model7'), GLOBAL.config.AXES_TPOINT_CONFIG_FILE_PATH_SUFFIX));
parts.model8.parts.configManager.configure(
    editableConfigAddress       := ADR(parts.model8.editableConfig),
    activeConfigAddress         := ADR(parts.model8.config),
    configLength                := SIZEOF(parts.model8.editableConfig),
    editableConfigSymbolName    := CONCAT(CONCAT(GLOBAL.config.AXES_TPOINT_EDITABLE_CONFIG_SYMBOL_PREFIX, 'model8'), GLOBAL.config.AXES_TPOINT_EDITABLE_CONFIG_SYMBOL_SUFFIX),
    activeConfigSymbolName      := CONCAT(CONCAT(GLOBAL.config.AXES_TPOINT_ACTIVE_CONFIG_SYMBOL_PREFIX, 'model8'), GLOBAL.config.AXES_TPOINT_ACTIVE_CONFIG_SYMBOL_SUFFIX),
    configFilePath              := CONCAT(CONCAT(GLOBAL.config.AXES_TPOINT_CONFIG_FILE_PATH_PREFIX, 'model8'), GLOBAL.config.AXES_TPOINT_CONFIG_FILE_PATH_SUFFIX));
parts.model9.parts.configManager.configure(
    editableConfigAddress       := ADR(parts.model9.editableConfig),
    activeConfigAddress         := ADR(parts.model9.config),
    configLength                := SIZEOF(parts.model9.editableConfig),
    editableConfigSymbolName    := CONCAT(CONCAT(GLOBAL.config.AXES_TPOINT_EDITABLE_CONFIG_SYMBOL_PREFIX, 'model9'), GLOBAL.config.AXES_TPOINT_EDITABLE_CONFIG_SYMBOL_SUFFIX),
    activeConfigSymbolName      := CONCAT(CONCAT(GLOBAL.config.AXES_TPOINT_ACTIVE_CONFIG_SYMBOL_PREFIX, 'model9'), GLOBAL.config.AXES_TPOINT_ACTIVE_CONFIG_SYMBOL_SUFFIX),
    configFilePath              := CONCAT(CONCAT(GLOBAL.config.AXES_TPOINT_CONFIG_FILE_PATH_PREFIX, 'model9'), GLOBAL.config.AXES_TPOINT_CONFIG_FILE_PATH_SUFFIX));
END_METHOD

METHOD _onFirstStart
VAR_INPUT
END_VAR
CASE _onFirstStartCurrentAction OF
    0:
        // start loading the config from XML file
        parts.model0.parts.configManager.processes.load.start(parts.model0.parts.configManager.processes.load.set.filePath);
        parts.model1.parts.configManager.processes.load.start(parts.model1.parts.configManager.processes.load.set.filePath);
        parts.model2.parts.configManager.processes.load.start(parts.model2.parts.configManager.processes.load.set.filePath);
        parts.model3.parts.configManager.processes.load.start(parts.model3.parts.configManager.processes.load.set.filePath);
        parts.model4.parts.configManager.processes.load.start(parts.model4.parts.configManager.processes.load.set.filePath);
        parts.model5.parts.configManager.processes.load.start(parts.model5.parts.configManager.processes.load.set.filePath);
        parts.model6.parts.configManager.processes.load.start(parts.model6.parts.configManager.processes.load.set.filePath);
        parts.model7.parts.configManager.processes.load.start(parts.model7.parts.configManager.processes.load.set.filePath);
        parts.model8.parts.configManager.processes.load.start(parts.model8.parts.configManager.processes.load.set.filePath);
        parts.model9.parts.configManager.processes.load.start(parts.model9.parts.configManager.processes.load.set.filePath);
        _onFirstStartCurrentAction := 1;
    1:
        // wait until the config has been loaded
        IF     parts.model0.parts.configManager.processes.load.statuses.busyStatus.idle
           AND parts.model1.parts.configManager.processes.load.statuses.busyStatus.idle 
           AND parts.model2.parts.configManager.processes.load.statuses.busyStatus.idle 
           AND parts.model3.parts.configManager.processes.load.statuses.busyStatus.idle 
           AND parts.model4.parts.configManager.processes.load.statuses.busyStatus.idle 
           AND parts.model5.parts.configManager.processes.load.statuses.busyStatus.idle 
           AND parts.model6.parts.configManager.processes.load.statuses.busyStatus.idle 
           AND parts.model7.parts.configManager.processes.load.statuses.busyStatus.idle 
           AND parts.model8.parts.configManager.processes.load.statuses.busyStatus.idle 
           AND parts.model9.parts.configManager.processes.load.statuses.busyStatus.idle 
        THEN
            // some files may have failed to load, because not all models may be present
            _onFirstStartCurrentAction := 2;
        END_IF
    2:
        // now start activating the configs
        parts.model0.parts.configManager.processes.activate.start();
        parts.model1.parts.configManager.processes.activate.start();
        parts.model2.parts.configManager.processes.activate.start();
        parts.model3.parts.configManager.processes.activate.start();
        parts.model4.parts.configManager.processes.activate.start();
        parts.model5.parts.configManager.processes.activate.start();
        parts.model6.parts.configManager.processes.activate.start();
        parts.model7.parts.configManager.processes.activate.start();
        parts.model8.parts.configManager.processes.activate.start();
        parts.model9.parts.configManager.processes.activate.start();
        _onFirstStartCurrentAction := 3;
    3:
        // wait until the configs have been activated
        IF      parts.model0.parts.configManager.processes.activate.statuses.busyStatus.idle 
            AND parts.model1.parts.configManager.processes.activate.statuses.busyStatus.idle 
            AND parts.model2.parts.configManager.processes.activate.statuses.busyStatus.idle 
            AND parts.model3.parts.configManager.processes.activate.statuses.busyStatus.idle 
            AND parts.model4.parts.configManager.processes.activate.statuses.busyStatus.idle 
            AND parts.model5.parts.configManager.processes.activate.statuses.busyStatus.idle 
            AND parts.model6.parts.configManager.processes.activate.statuses.busyStatus.idle 
            AND parts.model7.parts.configManager.processes.activate.statuses.busyStatus.idle 
            AND parts.model8.parts.configManager.processes.activate.statuses.busyStatus.idle 
            AND parts.model9.parts.configManager.processes.activate.statuses.busyStatus.idle 
        THEN
            _onFirstStartCurrentAction := 1000;
        END_IF
    999:
        // error, but nothing we can do about it now!
        ;
    1000:
        ; // nothing to do, done

END_CASE
END_METHOD

END_FUNCTION_BLOCK

// ---- MTCS/Axes/StateMachines/AxesAzimuthAxis.TcPOU
FUNCTION_BLOCK AxesAzimuthAxis EXTENDS SM_AxesAzimuthAxis
VAR_INPUT
END_VAR
VAR_OUTPUT
END_VAR
VAR_IN_OUT
END_VAR
VAR
    // setpoint generators
	{attribute 'OPC.UA.DA' := '0'}
    _aziSetGen : AxesExternalSetpointGenerator;
	{attribute 'OPC.UA.DA' := '0'}
    _ablSetGen : AxesTorqueSetpointGenerator;
    
    // helpers
	{attribute 'OPC.UA.DA' := '0'}
    _powerOnHelper : AxesPowerOnHelper;
	{attribute 'OPC.UA.DA' := '0'}
    _powerOffHelper : AxesPowerOffHelper;
	{attribute 'OPC.UA.DA' := '0'}
    _moveOutOfLimitSwitchHelper : AxesMoveOutOfLimitSwitchHelper;
	{attribute 'OPC.UA.DA' := '0'}
    _homingHelper : AxesHomingHelper;
	{attribute 'OPC.UA.DA' := '0'}
    _stopHelper : AxesStopHelper;
	{attribute 'OPC.UA.DA' := '0'}
    _quickStopHelper : AxesQuickStopHelper;
	{attribute 'OPC.UA.DA' := '0'}
    _setPositionHelper : AxesSetPositionHelper;
	{attribute 'OPC.UA.DA' := '0'}
    _unlockBrakeHelper : AxesUnlockBrakeHelper;
    
    // RMS and average setpoint deviation calculator
	{attribute 'OPC.UA.DA' := '0'}
    _deviationCalculator: AverageAndRmsCalculator;
    // local copy of the isTracking flag
	{attribute 'OPC.UA.DA' := '0'}
    _isTracking: BOOL;
END_VAR

_update();

_resetting();

_powerOnHelper(
    id                      := id,
    setpointGenerator       := _aziSetGen,
    powerOn                 := processes.powerOn,
    stop                    := processes.stop,
    reset                   := processes.reset,
    virtual                 := parts.virtualAxis,
    physical                := parts.physicalAxis,
    targetStart             := targetStart,
    pAblAxis                := ADR(parts.ablAxis),
    pAblDriveChannel        := ADR(ablDriveChannel),
    pAblSetpointGenerator   := ADR(_ablSetGen));
    
_powerOffHelper(
    setpointGenerator       := _aziSetGen,
    powerOff                := processes.powerOff,
    stop                    := processes.stop,
    virtual                 := parts.virtualAxis,
    physical                := parts.physicalAxis,
    pAblAxis                := ADR(parts.ablAxis),
    pAblDriveChannel        := ADR(ablDriveChannel),
    pAblSetpointGenerator   := ADR(_ablSetGen));

_moveOutOfLimitSwitchHelper(
    setpointGenerator            := _aziSetGen,
    positiveLimitSwitchError     := positiveLimitSwitchError,
    negativeLimitSwitchError     := negativeLimitSwitchError,
    positiveLimitSwitchInput     := config.positiveLimitSwitchInput,
    negativeLimitSwitchInput     := config.negativeLimitSwitchInput,
    moveOutOfLimitSwitchDistance := config.moveOutOfLimitSwitchDistance,
    moveOutOfLimitSwitch         := processes.moveOutOfLimitSwitch,
    moveRelative                 := processes.moveRelative,
    powerOn                      := processes.powerOn,
    reset                        := processes.reset,
    virtual                      := parts.virtualAxis,
    physical                     := parts.physicalAxis,
    driveChannel                 := aziMainDriveChannel);

_homingHelper(
    id                          := id,
    homingStartAbsEncPosition   := config.homingStartAbsEncPosition,
    homingVelocity              := config.homingVelocity,
    homingRange                 := config.homingRange,
    homingGotoStartVelocity     := config.homingGotoStartVelocity,
    homingHomePosition          := config.homingHomePosition,
    lidasInvert                 := config.lidasInvert,
    absoluteEncoderPosition     := absoluteEncoderPosition.degrees.value,
    lidaAveragePosition         := lidaAveragePosition.degrees.value,
    lida1Position               := lida1Position.degrees.value,
    setpointGenerator           := _aziSetGen,
    doHoming                    := processes.doHoming,
    stop                        := processes.stop,
    setPosition                 := processes.setPosition,
    virtual                     := parts.virtualAxis,
    physical                    := parts.physicalAxis,
    pLida1                      := ADR(parts.lida1),
    pLida2                      := ADR(parts.lida2),
    pLida3                      := ADR(parts.lida3),
    pLida4                      := ADR(parts.lida4));
    
_moveAbsolute();
_moveRelative();
_moveVelocity();
    
_stopHelper(
    setpointGenerator   := _aziSetGen,
    stop                := processes.stop,
    virtual             := parts.virtualAxis,
    physical            := parts.physicalAxis);
    
_quickStopHelper(
    deceleration        := config.quickStopDeceleration, 
    jerk                := config.quickStopJerk,
    setpointGenerator   := _aziSetGen,
    quickStop           := processes.quickStop,
    virtual             := parts.virtualAxis,
    physical            := parts.physicalAxis);
    
_setPositionHelper(
    setpointGenerator   := _aziSetGen,
    setPosition         := processes.setPosition,
    virtual             := parts.virtualAxis,
    physical            := parts.physicalAxis);
    
_unlockBrakeHelper(
    unlockBrake         := processes.unlockBrake,
    driveChannel        := aziDriveChannel);

_update();

METHOD callOnce : BOOL
VAR_INPUT
    dcTime : LINT; 
	targetPosDeg  : LREAL; // degrees
	targetVeloDegPerSec : LREAL; // degrees/sec
	targetAccDegPerSec2  : LREAL; // degrees/sec2
    trackingStart : LREAL; // degrees
    modelDelta : LREAL; // degrees
END_VAR
VAR_IN_OUT
    isTracking : BOOL;
END_VAR
VAR
END_VAR
// run the setpoint generators
_ablSetGen(
    ablMaxTorqueRiseSpeed   := config.ablMaxTorqueRiseSpeed,
    ablMaxTorqueFallSpeed   := config.ablMaxTorqueFallSpeed,
    maxAccelerationSetpoint := config.maxAccelerationSetpoint,
    ablMaxTorque            := config.ablMaxTorque,
    ablMinTorque            := config.ablMinTorque,
    ablZeroAccTorque        := config.ablZeroAccTorque,
    ablTorqueOutputOverride := config.ablTorqueOutputOverride,
    aziAndAblSameDirection  := config.aziAndAblSameDirection,
    ablPositiveTorque       := config.ablPositiveTorque,
    physicalAxis            := parts.physicalAxis,
    virtualAxis             := parts.virtualAxis,
    ablAxis                 := parts.ablAxis);
_aziSetGen( 
    dcTime                      := dcTime,
    tracking                    := isTracking,
    virtual                     := parts.virtualAxis.axis_ref, 
    physical                    := parts.physicalAxis.axis_ref, 
    targetPos                   := targetPosDeg, 
    targetVelo                  := targetVeloDegPerSec, 
    targetAcc                   := targetAccDegPerSec2, 
    trackingStart               := trackingStart,
    velocityLimit               := config.velocityLimit,
    accelerationLimit           := config.accelerationLimit,
    minTrackingPositionSetpoint := config.minPositionSetpoint,
    maxTrackingPositionSetpoint := config.maxPositionSetpoint,
    minVirtualPositionSetpoint  := config.minPositionLimitVirtualAxis,
    maxVirtualPositionSetpoint  := config.maxPositionLimitVirtualAxis,
    limitReached                => setPosLimitReached);
    
// update the torque command value
ablDriveChannel.torqueCommandValue := AxesCalculateTorqueCommandValue(
    torqueSetpoint := _ablSetGen.output / 180.0,
    torqueConstant := ablDriveChannel.torqueConstant,
    channelPeakCurrent := ablDriveChannel.channelPeakCurrent.amps.value);

// apply the position correction
IF parts.physicalAxis.axis_ref.Status.Homed THEN
    parts.physicalAxis.setPositionCorrection( -(lidaAveragePosition.degrees.value - parts.physicalAxis.axis_ref.NcToPlc.ActPosWithoutPosCorrection) );
ELSE
    parts.physicalAxis.setPositionCorrection(0.0);
END_IF

// calculate the average and RMS deviation
_deviationCalculator(in := parts.physicalAxis.axis_ref.NcToPlc.ActPos - parts.physicalAxis.axis_ref.NcToPlc.SetPos );
deviation1SecAverage(newDegreesValue := _deviationCalculator.avg);
deviation1SecRMS(newDegreesValue := _deviationCalculator.rms);

// keep a local copy of the isTracking variable
_isTracking := isTracking;
END_METHOD

METHOD _resetting : LREAL
VAR_INPUT
END_VAR
IF processes.reset.isBusy() THEN
    
    IF NOT processes.reset.isStarted() THEN
        processes.reset._state := 0;
        processes.reset.setStarted();
	END_IF
    
    CASE processes.reset._state OF
        0:
            // reset all processes so that they are green again
            processes.doHoming.resetIfIdle();
            processes.moveAbsolute.resetIfIdle();
            processes.moveOutOfLimitSwitch.resetIfIdle();
            processes.moveRelative.resetIfIdle();
            processes.moveVelocity.resetIfIdle();
            processes.powerOff.resetIfIdle();
            processes.powerOn.resetIfIdle();
            processes.quickStop.resetIfIdle();
            processes.setPosition.resetIfIdle();
            processes.stop.resetIfIdle();
            processes.unlockBrake.resetIfIdle();
            
            processes.reset.setActualStatus('Powering off the axis');
            // power off the axis
            processes.powerOff.start();
            processes.reset._state := 1;
        1:
            IF processes.powerOff.isIdle() THEN
                // regardless of whether power off worked or not, proceed    
                processes.reset._state := 2;
			END_IF
        2:
            // update the physical axis soft position limit values
            parts.physicalAxis.processes.writeParameter.start(parameterNumber := MC_AxisParameter.SWLimitNeg, value := config.minPositionLimitPhysicalAxis);
            processes.reset._state := 3;
        3:
            IF parts.physicalAxis.processes.writeParameter.isIdle() THEN
                IF parts.physicalAxis.processes.writeParameter.isGood() THEN
                    processes.reset._state := 4;
                ELSE
                    processes.reset.setActualStatus(CONCAT('Could not set the physical SWLimitNeg: ', parts.physicalAxis.processes.writeParameter.actualStatus));
                    processes.reset._state := 999;
				END_IF
			END_IF
        4:
            parts.physicalAxis.processes.writeParameter.start(parameterNumber := MC_AxisParameter.SWLimitPos, value := config.maxPositionLimitPhysicalAxis);
            processes.reset._state := 5;
        5:
            IF parts.physicalAxis.processes.writeParameter.isIdle() THEN
                IF parts.physicalAxis.processes.writeParameter.isGood() THEN
                    processes.reset._state := 6;
                ELSE
                    processes.reset.setActualStatus(CONCAT('Could not set the physical SWLimitPos: ', parts.physicalAxis.processes.writeParameter.actualStatus));
                    processes.reset._state := 999;
				END_IF
			END_IF
        6:
            parts.physicalAxis.processes.writeBoolParameter.start(parameterNumber := MC_AxisParameter.EnableLimitNeg, value := TRUE);
            processes.reset._state := 7;
        7:
            IF parts.physicalAxis.processes.writeBoolParameter.isIdle() THEN
                IF parts.physicalAxis.processes.writeBoolParameter.isGood() THEN
                    processes.reset._state := 8;
                ELSE
                    processes.reset.setActualStatus(CONCAT('Could not set the physical EnableLimitNeg: ', parts.physicalAxis.processes.writeBoolParameter.actualStatus));
                    processes.reset._state := 999;
				END_IF
			END_IF
        8:
            parts.physicalAxis.processes.writeBoolParameter.start(parameterNumber := MC_AxisParameter.EnableLimitPos, value := TRUE);
            processes.reset._state := 9;
        9:
            IF parts.physicalAxis.processes.writeBoolParameter.isIdle() THEN
                IF parts.physicalAxis.processes.writeBoolParameter.isGood() THEN
                    processes.reset._state := 10;
                ELSE
                    processes.reset.setActualStatus(CONCAT('Could not set the physical EnableLimitPos: ', parts.physicalAxis.processes.writeBoolParameter.actualStatus));
                    processes.reset._state := 999;
				END_IF
			END_IF
        10:
            // update the virtual axis soft position limit values
            parts.virtualAxis.processes.writeParameter.start(parameterNumber := MC_AxisParameter.SWLimitNeg, value := config.minPositionLimitVirtualAxis);
            processes.reset._state := 11;
        11:
            IF parts.virtualAxis.processes.writeParameter.isIdle() THEN
                IF parts.virtualAxis.processes.writeParameter.isGood() THEN
                    processes.reset._state := 12;
                ELSE
                    processes.reset.setActualStatus(CONCAT('Could not set the virtual SWLimitNeg: ', parts.virtualAxis.processes.writeParameter.actualStatus));
                    processes.reset._state := 999;
				END_IF
			END_IF
        12:
            parts.virtualAxis.processes.writeParameter.start(parameterNumber := MC_AxisParameter.SWLimitPos, value := config.maxPositionLimitVirtualAxis);
            processes.reset._state := 13;
        13:
            IF parts.virtualAxis.processes.writeParameter.isIdle() THEN
                IF parts.virtualAxis.processes.writeParameter.isGood() THEN
                    processes.reset._state := 14;
                ELSE
                    processes.reset.setActualStatus(CONCAT('Could not set the virtual SWLimitPos: ', parts.virtualAxis.processes.writeParameter.actualStatus));
                    processes.reset._state := 999;
				END_IF
			END_IF
        14:
            parts.virtualAxis.processes.writeBoolParameter.start(parameterNumber := MC_AxisParameter.EnableLimitNeg, value := TRUE);
            processes.reset._state := 15;
        15:
            IF parts.virtualAxis.processes.writeBoolParameter.isIdle() THEN
                IF parts.virtualAxis.processes.writeBoolParameter.isGood() THEN
                    processes.reset._state := 16;
                ELSE
                    processes.reset.setActualStatus(CONCAT('Could not set the virtual EnableLimitNeg: ', parts.virtualAxis.processes.writeBoolParameter.actualStatus));
                    processes.reset._state := 999;
				END_IF
			END_IF
        16:
            parts.virtualAxis.processes.writeBoolParameter.start(parameterNumber := MC_AxisParameter.EnableLimitPos, value := TRUE);
            processes.reset._state := 17;
        17:
            IF parts.virtualAxis.processes.writeBoolParameter.isIdle() THEN
                IF parts.virtualAxis.processes.writeBoolParameter.isGood() THEN
                    processes.reset._state := 18;
                ELSE
                    processes.reset.setActualStatus(CONCAT('Could not set the virtual EnableLimitPos: ', parts.virtualAxis.processes.writeBoolParameter.actualStatus));
                    processes.reset._state := 999;
				END_IF
			END_IF
        18:
            // unlock the ABL motor brake
            ablDriveChannel.processes.setBrake.start(newState := DriveBrakeStates.BRAKE_FORCE_UNLOCK);
            processes.reset._state := 19;
        19:
            IF ablDriveChannel.processes.setBrake.isIdle() THEN
                IF ablDriveChannel.processes.setBrake.isGood() THEN
                    processes.reset._state := 20;
                ELSE
                    processes.reset.setActualStatus('Could not unlock the ABL motor brake!');
                    processes.reset._state := 999;
				END_IF
			END_IF
        20:
            // try to acknowledge the safe state (if present)
            processes.reset.setActualStatus('Resetting safety');
            aziDriveChannel.processes.acknowledgeSafetyError.start();
            ablDriveChannel.processes.acknowledgeSafetyError.start();
            processes.reset._state := 21;
        21:
            IF aziDriveChannel.processes.acknowledgeSafetyError.isIdle() AND ablDriveChannel.processes.acknowledgeSafetyError.isIdle()  THEN
                IF aziDriveChannel.processes.acknowledgeSafetyError.isGood() AND ablDriveChannel.processes.acknowledgeSafetyError.isGood() THEN
                    processes.reset._state := 22;
                ELSE
                    processes.reset.setActualStatus('Cannot get out of safe state!');
                    processes.reset._state := 999;
                END_IF
            END_IF
        22:
            // reset the drive channel
            processes.reset.setActualStatus('Resetting the drive channel');
            aziDriveChannel.processes.reset.start();
            ablDriveChannel.processes.reset.start();
            processes.reset._state := 23;
        23:
            IF aziDriveChannel.processes.reset.isIdle() AND ablDriveChannel.processes.reset.isIdle() THEN
                IF aziDriveChannel.processes.reset.isGood() AND ablDriveChannel.processes.reset.isGood() THEN
                    processes.reset._state := 24;
                ELSE
                    processes.reset.setActualStatus('Could not reset the drive channels!');
                    processes.reset._state := 999;
                END_IF
            END_IF
        24:
            // update the drive channel
            processes.reset.setActualStatus('Updating the drive channel');
            aziDriveChannel.processes.update.start();
            ablDriveChannel.processes.update.start();
            processes.reset._state := 25;
        25:
            IF aziDriveChannel.processes.update.isIdle() AND ablDriveChannel.processes.update.isIdle() THEN
                IF aziDriveChannel.processes.update.isGood() AND ablDriveChannel.processes.update.isGood() THEN
                    processes.reset._state := 26;
                ELSE
                    processes.reset.setActualStatus('Could not update the drive channel!');
                    processes.reset._state := 999;
                END_IF
            END_IF
        26:
            // reset the axis
            processes.reset.setActualStatus('Resetting the axes');
            parts.physicalAxis.processes.reset.start();
            parts.ablAxis.processes.reset.start();
            parts.virtualAxis.processes.reset.start();
            processes.reset._state := 27;
        27:
            IF     parts.virtualAxis.processes.reset.isIdle() 
               AND parts.physicalAxis.processes.reset.isIdle() 
               AND parts.ablAxis.processes.reset.isIdle() THEN
                IF     parts.virtualAxis.processes.reset.isGood() 
                   AND parts.physicalAxis.processes.reset.isGood() 
                   AND parts.ablAxis.processes.reset.isGood() THEN
                    processes.reset._state := 28;
                ELSE
                    processes.reset.setActualStatus('Could not reset the axes');
                    processes.reset._state := 999;
                END_IF
            END_IF
        28:
            // synchronize the motor encoder with the absolute encoder, if we haven't homed
            IF parts.physicalAxis.axis_ref.Status.Homed THEN
                processes.reset._state := 1000;
            ELSE
                parts.physicalAxis.processes.setPosition.start(value := absoluteEncoderPosition.degrees.value);
                processes.reset._state := 29;
			END_IF
        29:
            IF parts.physicalAxis.processes.setPosition.isIdle() THEN
                IF parts.physicalAxis.processes.setPosition.isGood() THEN
                    processes.reset._state := 1000;
                ELSE
                    processes.reset.setActualStatus('Could not sync motor enc with abs enc');
                    processes.reset._state := 999;
				END_IF
			END_IF
        999:
            // error!
            processes.reset.setBad();
            processes.reset.setFinished();
        1000:
            processes.reset.setActualStatus('Reset done');
            // ok done
            processes.reset.setFinished();
            processes.reset.setGood();
    END_CASE
    
END_IF
END_METHOD

METHOD _moveRelative
VAR_INPUT
END_VAR
VAR
    distanceDegrees : LREAL;
END_VAR
IF processes.moveRelative.isBusy() THEN
    
    IF NOT processes.moveRelative.isStarted() THEN
        
        distanceDegrees := AxesMoveUnitsToDeg(units := processes.moveRelative.get.units, value := processes.moveRelative.get.value);
        
        parts.virtualAxis.processes.moveRelative.start(distance := distanceDegrees, maxVelocity := config.maxVelocitySetpoint);
    
        processes.moveRelative.setStarted();
    ELSE
        
        // update the statuses
        processes.moveRelative.statuses.healthStatus(
            isGood := parts.virtualAxis.processes.moveRelative.statuses.healthStatus.isGood,
            hasWarning := parts.virtualAxis.processes.moveRelative.statuses.healthStatus.hasWarning);
        processes.moveRelative.setActualStatus(parts.virtualAxis.processes.moveRelative.actualStatus);
        processes.moveRelative.statuses.busyStatus(isBusy := parts.virtualAxis.processes.moveRelative.statuses.busyStatus.isBusy);
    
	END_IF
END_IF
END_METHOD

METHOD _moveVelocity
VAR_INPUT
END_VAR
VAR
    velocityDegPerSec : LREAL;
END_VAR
IF processes.moveVelocity.isBusy() THEN
    
    IF NOT processes.moveVelocity.isStarted() THEN
        
        velocityDegPerSec := AxesMoveVelocityUnitsToDegPerSec(units := processes.moveVelocity.get.units, value := processes.moveVelocity.get.value);
        
        parts.virtualAxis.processes.moveVelocity.start(value := velocityDegPerSec);
    
        processes.moveVelocity.setStarted();
            
	END_IF

    // update the statuses
    processes.moveVelocity.statuses.busyStatus(isBusy := parts.virtualAxis.processes.moveVelocity.statuses.busyStatus.isBusy);
    processes.moveVelocity.statuses.healthStatus(
        isGood := parts.virtualAxis.processes.moveVelocity.statuses.healthStatus.isGood,
        hasWarning := parts.virtualAxis.processes.moveVelocity.statuses.healthStatus.hasWarning);
    processes.moveVelocity.setActualStatus(parts.virtualAxis.processes.moveVelocity.actualStatus);

END_IF
END_METHOD

METHOD _moveAbsolute
VAR_INPUT
END_VAR
VAR
END_VAR
IF processes.moveAbsolute.isBusy() THEN
    
    IF NOT processes.moveAbsolute.isStarted() THEN
        
    
        targetStart(newDegreesValue := AxesMoveUnitsToDeg(units := processes.moveAbsolute.get.units, value := processes.moveAbsolute.get.value));
        
        parts.virtualAxis.processes.moveAbsolute.start(position := targetStart.degrees.value + processes.moveAbsolute.get.offset, maxVelocity := config.maxVelocitySetpoint);

        processes.moveAbsolute.setStarted();
        
    END_IF

    IF parts.virtualAxis.processes.moveAbsolute.isIdle() THEN
        
        IF parts.virtualAxis.processes.moveAbsolute.isGood() THEN
            processes.moveAbsolute.setGood();
        ELSE
            processes.moveAbsolute.setBad();
		END_IF
        
        processes.moveAbsolute.setActualStatus(parts.virtualAxis.processes.moveAbsolute.actualStatus);
        processes.moveAbsolute.setFinished();
    
	END_IF
    
END_IF
END_METHOD

METHOD _update : LREAL
VAR_INPUT
END_VAR
VAR
    absoluteEncoderReduction : LREAL;
END_VAR
// update the superclass
SUPER^(
    config := config,
    aziDriveChannel := aziDriveChannel,
    ablDriveChannel := ablDriveChannel,
    aziMainDriveChannel := aziMainDriveChannel,
    ablMainDriveChannel := ablMainDriveChannel);
    
// update the limit switches
positiveLimitSwitchError := NOT GETBIT32(inVal32 := INT_TO_DWORD(aziMainDriveChannel.digitalInputs), bitNo := config.positiveLimitSwitchInput);
negativeLimitSwitchError := NOT GETBIT32(inVal32 := INT_TO_DWORD(aziMainDriveChannel.digitalInputs), bitNo := config.negativeLimitSwitchInput);

// update the LIDA positions
lida1Position(newDegreesValue := AxesLidaValueToPosition(id := AxesIds.AZI, encoderValue := parts.lida1.counterValue, invert := config.lidasInvert));
lida2Position(newDegreesValue := AxesLidaValueToPosition(id := AxesIds.AZI, encoderValue := parts.lida2.counterValue, invert := config.lidasInvert));
lida3Position(newDegreesValue := AxesLidaValueToPosition(id := AxesIds.AZI, encoderValue := parts.lida3.counterValue, invert := config.lidasInvert));
lida4Position(newDegreesValue := AxesLidaValueToPosition(id := AxesIds.AZI, encoderValue := parts.lida4.counterValue, invert := config.lidasInvert));

// calculate the average value
lidaAveragePosition( newDegreesValue := 
    AxesCalculateLidaAveragePosition(
        lida1Position := lida1Position.degrees.value,
        lida2Position := lida2Position.degrees.value,
        lida3Position := lida3Position.degrees.value,
        lida4Position := lida4Position.degrees.value,
        useLida1      := NOT (parts.lida1.openCircuit OR parts.lida1.syncError OR parts.lida1.extrapolationStall), 
        useLida2      := NOT (parts.lida2.openCircuit OR parts.lida2.syncError OR parts.lida2.extrapolationStall), 
        useLida3      := NOT (parts.lida3.openCircuit OR parts.lida3.syncError OR parts.lida3.extrapolationStall), 
        useLida4      := NOT (parts.lida4.openCircuit OR parts.lida4.syncError OR parts.lida4.extrapolationStall)));

// update the absolute encoder position
IF  config.absoluteEncoderInvert THEN
    absoluteEncoderReduction := -REDUCTION_ABS_ENC_TO_TEL;
ELSE
    absoluteEncoderReduction := REDUCTION_ABS_ENC_TO_TEL;
END_IF
absoluteEncoderPosition(newDegreesValue := AxesSSIValueToPosition(
        reduction       := absoluteEncoderReduction,
        encoderValue    := parts.absoluteEncoder.counterValue,
        zeroOffset      := config.absoluteEncoderOffset));

// update the position/velocity/acceleration
actPos(newDegreesValue := parts.physicalAxis.axis_ref.NcToPlc.ActPos);
actVelo(newDegreesPerSecondValue := parts.physicalAxis.axis_ref.NcToPlc.ActVelo);
actAcc(newDegreesPerSquareSecondValue := parts.physicalAxis.axis_ref.NcToPlc.ActAcc);
setPos(newDegreesValue := parts.physicalAxis.axis_ref.NcToPlc.SetPos);
setVelo(newDegreesPerSecondValue := parts.physicalAxis.axis_ref.NcToPlc.SetVelo);
setAcc(newDegreesPerSquareSecondValue := parts.physicalAxis.axis_ref.NcToPlc.SetAcc);
IF parts.physicalAxis.axis_ref.Status.ExtSetPointGenEnabled THEN
    targetPos(newDegreesValue := parts.physicalAxis.axis_ref.PlcToNc.ExtSetPos);
    targetOffset(newDegreesValue := parts.virtualAxis.actPos.degrees.value - targetStart.degrees.value);
ELSE
    targetPos(newDegreesValue := parts.physicalAxis.axis_ref.NcToPlc.TargetPos);
    targetOffset(newDegreesValue := 0.0);
END_IF

// update the actual torque feedback on the telescope side
actTorqueAzi(newNewtonmeterValue := aziDriveChannel.actualTorqueFeedback.newtonmeter.value * REDUCTION_AZI_TO_TEL);
actTorqueAbl(newNewtonmeterValue := ablDriveChannel.actualTorqueFeedback.newtonmeter.value * REDUCTION_ABL_TO_TEL);


// check if the motor is slipping w.r.t. the lidas
slipError :=     parts.physicalAxis.axis_ref.Status.Homed 
             AND parts.physicalAxis.axis_ref.Status.ExtSetPointGenEnabled 
             AND (ABS(parts.physicalAxis.axis_ref.PlcToNc.PositionCorrection) > config.slipLimit);
END_METHOD

END_FUNCTION_BLOCK

// ---- MTCS/Axes/StateMachines/AxesPointingModelSetup.TcPOU
FUNCTION_BLOCK AxesPointingModelSetup EXTENDS SM_AxesPointingModelSetup
VAR_INPUT
END_VAR
VAR_OUTPUT
END_VAR
VAR
	{attribute 'OPC.UA.DA' := '0'}
    _testVar : BOOL; // without any variable, the superclass attributes are not visible in the UA address space
END_VAR

SUPER^();

END_FUNCTION_BLOCK

// ---- MTCS/Axes/StateMachines/AxesTarget.TcPOU
FUNCTION_BLOCK AxesTarget EXTENDS SM_AxesTarget
VAR_INPUT
END_VAR
VAR_OUTPUT
END_VAR
VAR
END_VAR

SUPER^();

METHOD updateAziEle
VAR_INPUT
	input : TmcAzElFull; // units: see SLALIB AltAz
    deltaAzi : LREAL := 0; // arcseconds
    deltaEle : LREAL := 0; // arcseconds
END_VAR
// formulas: see SLALIB documentation: slaAltaz 

(* Natural units are used throughout. The arguments ha, dec, phi, az, el AND zd are in
radians. The velocities and accelerations assume constant declination and constant
rate of change of hour angle (as for tracking a star); the units of azd, eld and pad
are radians per radian of HA, while the units of azdd, eldd and padd are radians per
radian of HA squared. To convert into practical degree- and second-based units:
 angles * 360/2pi                          --> degrees
 velocities *(2pi/86400) * (360/2pi)       --> degree/sec
 accelerations * (2pi/86400)^2 * (360/2pi) --> degree/sec/sec
*)

aziPointingModelOffset(newDegreesValue := ARCSEC_TO_DEG(deltaAzi));
elePointingModelOffset(newDegreesValue := ARCSEC_TO_DEG(deltaEle));

aziPos(newDegreesValue := RAD_TO_DEG(input.az) + aziPointingModelOffset.degrees.value);
aziVelo(newDegreesPerSecondValue := RAD_TO_DEG(input.azd  * (2*PI/86400.0)));
aziAcc(newDegreesPerSquareSecondValue := RAD_TO_DEG(input.azdd * (2*PI/86400.0) * (2*PI/86400.0)));

elePos(newDegreesValue := RAD_TO_DEG(input.el) + elePointingModelOffset.degrees.value);
eleVelo(newDegreesPerSecondValue := RAD_TO_DEG(input.eld  * (2*PI/86400.0)));
eleAcc(newDegreesPerSquareSecondValue := RAD_TO_DEG(input.eldd * (2*PI/86400.0) * (2*PI/86400.0)));

paPos(newDegreesValue := RAD_TO_DEG(input.pa));
paVelo(newDegreesPerSecondValue := RAD_TO_DEG(input.pad  * (2*PI/86400.0)));
paAcc(newDegreesPerSquareSecondValue := RAD_TO_DEG(input.padd * (2*PI/86400.0) * (2*PI/86400.0)));
END_METHOD

END_FUNCTION_BLOCK

// ---- MTCS/Axes/StateMachines/AxesFeedback.TcPOU
FUNCTION_BLOCK AxesFeedback EXTENDS SM_AxesFeedback
VAR_INPUT
END_VAR
VAR_OUTPUT
END_VAR
VAR
END_VAR

SUPER^();

END_FUNCTION_BLOCK

// ---- MTCS/Axes/Widgets/AxesAlphaWidget.TcPOU
FUNCTION_BLOCK AxesAlphaWidget
VAR_INPUT
    radians : LREAL;
END_VAR
VAR_OUTPUT
    hms : HoursMinutesSeconds;
    hours : LREAL;
    hmsString : STRING;
    
END_VAR
VAR
    _secondsTruncated : LREAL;
    _hmsFormat : STRING := '%dh %.2dm %04.1fs';
    _formatString : FB_FormatString;
END_VAR


hours := RAD_TO_HOUR(radians);


hms.positive:= radians > 0;
hms.hours   := TRUNC(ABS(hours));
hms.minutes := TRUNC( (ABS(hours) - hms.hours) * 60.0 );
hms.seconds := ((ABS(hours) - hms.hours) * 60.0 - hms.minutes) * 60.0;


_secondsTruncated := (LTRUNC(hms.seconds * 10.0) / 10.0 );

_formatString(
    sFormat := _hmsFormat,
    arg1 := F_DINT(hms.hours),
    arg2 := F_DINT(hms.minutes),
    arg3 := F_LREAL( _secondsTruncated ),
    sOut => hmsString);
    
IF NOT hms.positive THEN
    hmsString := CONCAT('-', hmsString);
END_IF

END_FUNCTION_BLOCK

// ---- MTCS/Axes/Widgets/AxesAngleWidget.TcPOU
FUNCTION_BLOCK AxesAngleWidget
VAR_INPUT
    degrees : LREAL;
    format : STRING := '%d° %.2d$' %04.1f"';
    showPlus : BOOL := FALSE;
    showMinus : BOOL := TRUE;
END_VAR
VAR_OUTPUT
    dms : DegreesMinutesSeconds;
    dmsString : STRING;    
END_VAR
VAR
    _secondsTruncated : LREAL;
    _formatString : FB_FormatString;
END_VAR


dms.positive:= degrees > 0;
dms.degrees := TRUNC(ABS(degrees));
dms.minutes := TRUNC( (ABS(degrees) - dms.degrees) * 60.0 );
dms.seconds := ((ABS(degrees) - dms.degrees) * 60.0 - dms.minutes) * 60.0;

_secondsTruncated := (LTRUNC(dms.seconds * 10.0) / 10.0 );
_formatString(
    sFormat := format,
    arg1 := F_DINT(dms.degrees),
    arg2 := F_DINT(dms.minutes),
    arg3 := F_LREAL( _secondsTruncated ),
    sOut => dmsString);

IF dms.positive THEN
    IF showPlus THEN
        dmsString := CONCAT('+', dmsString);
    END_IF;
ELSE
    IF showMinus THEN
        dmsString := CONCAT('-', dmsString);
    END_IF;
END_IF

END_FUNCTION_BLOCK

// ---- MTCS/Axes/Widgets/AxesPointRelativeProcessWidget.TcPOU
FUNCTION_BLOCK AxesPointRelativeProcessWidget
VAR_INPUT
    title : STRING;
    units : AxesMoveProcessWidgetUnits;
    
    actualStatus : StatusWidget;
    
    
    field_alpha_sign : AxesDialogSign;
    field_alpha_h : LREAL;
    field_alpha_m : LREAL;
    field_alpha_s : LREAL;
    field_alpha_decimal : LREAL;
    
    field_delta_sign : AxesDialogSign;
    field_delta_d : LREAL;
    field_delta_m : LREAL;
    field_delta_s : LREAL;
    field_delta_decimal : LREAL;
    
    field_roc_sign : AxesDialogSign;
    field_roc_d : LREAL;
    field_roc_m : LREAL;
    field_roc_s : LREAL;
    field_roc_decimal : LREAL;
    
    field_ron_sign : AxesDialogSign;
    field_ron_d : LREAL;
    field_ron_m : LREAL;
    field_ron_s : LREAL;
    field_ron_decimal : LREAL;
    
    alphaDisabled : BOOL;
    deltaDisabled : BOOL;
    rocDisabled : BOOL;
    ronDisabled : BOOL;
END_VAR
VAR_OUTPUT
    unitsText : STRING;
    alphaDeg : LREAL;
    deltaDeg : LREAL;
    rocDeg : LREAL;
    ronDeg : LREAL;
    
    
END_VAR
VAR_IN_OUT
    process : AxesPointRelativeProcess;
END_VAR
VAR
END_VAR


actualStatus(
    text  := process.actualStatus,
    color := HealthBusyToColor(healthStatus := process.statuses.healthStatus, 
                               busyStatus   := process.statuses.busyStatus));

CASE units OF
    AxesMoveProcessWidgetUnits.ARCMINUTES:
        unitsText := '$'';
        alphaDeg := field_alpha_decimal / 60.0;
        deltaDeg := field_delta_decimal / 60.0;
        rocDeg := field_roc_decimal / 60.0;
        ronDeg := field_ron_decimal / 60.0;
    AxesMoveProcessWidgetUnits.ARCSECCONDS:
        unitsText := '"';
        alphaDeg := field_alpha_decimal / 3600.0;
        deltaDeg := field_delta_decimal / 3600.0;
        rocDeg := field_roc_decimal / 3600.0;
        ronDeg := field_ron_decimal / 3600.0;
    AxesMoveProcessWidgetUnits.DEGMINSEC:
        unitsText := '';
        alphaDeg := HMS_TO_DEG(
            positive := field_alpha_sign = AxesDialogSign.DIALOG_PLUS,
            hours    := field_alpha_h,
            minutes  := field_alpha_m,
            seconds  := field_alpha_s);
        deltaDeg := DMS_TO_DEG(
            positive := field_delta_sign = AxesDialogSign.DIALOG_PLUS,
            degrees  := field_delta_d,
            minutes  := field_delta_m,
            seconds  := field_delta_s);
        rocDeg := DMS_TO_DEG(
            positive := field_roc_sign = AxesDialogSign.DIALOG_PLUS,
            degrees  := field_roc_d,
            minutes  := field_roc_m,
            seconds  := field_roc_s);
        ronDeg := DMS_TO_DEG(
            positive := field_ron_sign = AxesDialogSign.DIALOG_PLUS,
            degrees  := field_ron_d,
            minutes  := field_ron_m,
            seconds  := field_ron_s);
    AxesMoveProcessWidgetUnits.DEGREES:
        unitsText := '°';
        alphaDeg := field_alpha_decimal;
        deltaDeg := field_delta_decimal;
        rocDeg := field_roc_decimal;
        ronDeg := field_ron_decimal;
    AxesMoveProcessWidgetUnits.RADIANS:
        unitsText := 'rad';
        alphaDeg := RAD_TO_DEG(field_alpha_decimal);
        deltaDeg := RAD_TO_DEG(field_delta_decimal);
        rocDeg := RAD_TO_DEG(field_roc_decimal);
        ronDeg := RAD_TO_DEG(field_ron_decimal);
END_CASE

END_FUNCTION_BLOCK

// ---- MTCS/Common/Widgets/StatusWidget.TcPOU
FUNCTION_BLOCK StatusWidget
VAR_INPUT
	text  : STRING;
	color : StatusColor;
END_VAR
VAR_OUTPUT
END_VAR
VAR_IN_OUT
END_VAR
VAR
END_VAR

END_FUNCTION_BLOCK

// ---- MTCS/Common/HelperCode/HealthBusyToColor.TcPOU
FUNCTION HealthBusyToColor : StatusColor
VAR_IN_OUT
    healthStatus : HealthStatus;
    busyStatus   : BusyStatus;
END_VAR
VAR_OUTPUT
END_VAR
VAR
END_VAR

IF healthStatus.good THEN
	IF busyStatus.busy THEN
		HealthBusyToColor.fg := Colors.WHITE;
		HealthBusyToColor.bg := Colors.BLUE;
	ELSE
		HealthBusyToColor.fg := Colors.BLACK;
		HealthBusyToColor.bg := Colors.GREEN;
	END_IF
ELSIF healthStatus.bad THEN
	HealthBusyToColor.fg := Colors.WHITE;
	HealthBusyToColor.bg := Colors.RED;
ELSIF healthStatus.warning THEN
	HealthBusyToColor.fg := Colors.WHITE;
	HealthBusyToColor.bg := Colors.ORANGE;
ELSE
	HealthBusyToColor.fg := Colors.BLACK;
	HealthBusyToColor.bg := Colors.GRAY;
END_IF

END_FUNCTION

// ---- MTCS/Axes/Widgets/AxesDeltaWidget.TcPOU
FUNCTION_BLOCK AxesDeltaWidget
VAR_INPUT
    radians : LREAL;
END_VAR
VAR_OUTPUT
    dms : DegreesMinutesSeconds;
    degrees : LREAL;
    dmsString : STRING;    
END_VAR
VAR
    _secondsTruncated : LREAL;
    _dmsFormat : STRING := '%d° %.2d$' %04.1f"';
    _formatString : FB_FormatString;
END_VAR


degrees := RAD_TO_DEG(radians);

dms.positive:= radians > 0;
dms.degrees := TRUNC(ABS(degrees));
dms.minutes := TRUNC( (ABS(degrees) - dms.degrees) * 60.0 );
dms.seconds := ((ABS(degrees) - dms.degrees) * 60.0 - dms.minutes) * 60.0;



_secondsTruncated := (LTRUNC(dms.seconds * 10.0) / 10.0 );
_formatString(
    sFormat := _dmsFormat,
    arg1 := F_DINT(dms.degrees),
    arg2 := F_DINT(dms.minutes),
    arg3 := F_LREAL(_secondsTruncated),
    sOut => dmsString);

IF dms.positive THEN
    dmsString := CONCAT('+', dmsString);
ELSE
    dmsString := CONCAT('-', dmsString);
END_IF

END_FUNCTION_BLOCK

// ---- MTCS/Axes/Widgets/AxesManualJoystickAziEleWidget.TcPOU
FUNCTION_BLOCK AxesManualJoystickAziEleWidget
VAR_INPUT

    joystick_hold : BOOL := TRUE; 

    joystick_velocity_fast : LREAL := 3.0;   // degrees/s
    joystick_velocity_medium : LREAL := 1.0; // degrees/s
    joystick_velocity_slow : LREAL := 0.1;   // degrees/s
    
    jog_azi_forward_fast    : BOOL;
    jog_azi_forward_medium  : BOOL;
    jog_azi_forward_slow    : BOOL;
    jog_azi_backwards_fast    : BOOL;
    jog_azi_backwards_medium  : BOOL;
    jog_azi_backwards_slow    : BOOL;
    
    jog_ele_forward_fast    : BOOL;
    jog_ele_forward_medium  : BOOL;
    jog_ele_forward_slow    : BOOL;
    jog_ele_backwards_fast    : BOOL;
    jog_ele_backwards_medium  : BOOL;
    jog_ele_backwards_slow    : BOOL;
END_VAR
VAR_OUTPUT
    jog_azi_disabled : BOOL;
    jog_ele_disabled : BOOL;
    
    joystick_disabled : BOOL;
    
 
END_VAR
VAR_IN_OUT
    ref : Axes;
END_VAR
VAR
    aziJogForward : BOOL;
    aziJogBackwards : BOOL;
    aziJogVelocity : LREAL;
    eleJogForward : BOOL;
    eleJogBackwards : BOOL;
    eleJogVelocity : LREAL;
    
    aziJogForwardTrig : R_TRIG;
    aziJogBackwardsTrig : R_TRIG;
    eleJogForwardTrig : R_TRIG;
    eleJogBackwardsTrig : R_TRIG;
    
END_VAR

// azimuth
IF joystick_hold THEN
    jog_azi_disabled := (NOT ref.parts.azi.parts.virtualAxis.isJogEnabled) OR ref.parts.azi.statuses.poweredStatus.disabled;
ELSE
    jog_azi_disabled := ref.parts.azi.processes.moveVelocity.statuses.enabledStatus.disabled OR ref.parts.azi.statuses.poweredStatus.disabled;
END_IF

aziJogForward   := jog_azi_forward_fast OR jog_azi_forward_medium OR jog_azi_forward_slow;
aziJogBackwards := jog_azi_backwards_fast OR jog_azi_backwards_medium OR jog_azi_backwards_slow;
IF jog_azi_forward_fast OR jog_azi_backwards_fast THEN
    aziJogVelocity := joystick_velocity_fast;
ELSIF jog_azi_forward_medium OR jog_azi_backwards_medium THEN
    aziJogVelocity := joystick_velocity_medium;
ELSIF jog_azi_forward_slow OR jog_azi_backwards_slow THEN
    aziJogVelocity := joystick_velocity_slow;
END_IF

aziJogForwardTrig(CLK := aziJogForward);
aziJogBackwardsTrig(CLK := aziJogBackwards);

IF joystick_hold THEN
    ref.parts.azi.parts.virtualAxis.jog(aziJogForward, aziJogBackwards, aziJogVelocity, 0.0, 0.0);
ELSIF aziJogForwardTrig.Q THEN
    ref.parts.azi.processes.moveVelocity.request(units := AxesMoveVelocityUnits.DEGREES_PER_SECOND, aziJogVelocity);
ELSIF aziJogBackwardsTrig.Q THEN
    ref.parts.azi.processes.moveVelocity.request(units := AxesMoveVelocityUnits.DEGREES_PER_SECOND, -aziJogVelocity);
END_IF

// elevation
IF joystick_hold THEN
    jog_ele_disabled := (NOT ref.parts.ele.parts.virtualAxis.isJogEnabled) OR ref.parts.ele.statuses.poweredStatus.disabled;
ELSE
    jog_ele_disabled := ref.parts.ele.processes.moveVelocity.statuses.enabledStatus.disabled OR ref.parts.ele.statuses.poweredStatus.disabled;
END_IF

eleJogForward   := jog_ele_forward_fast OR jog_ele_forward_medium OR jog_ele_forward_slow;
eleJogBackwards := jog_ele_backwards_fast OR jog_ele_backwards_medium OR jog_ele_backwards_slow;
IF jog_ele_forward_fast OR jog_ele_backwards_fast THEN
    eleJogVelocity := joystick_velocity_fast;
ELSIF jog_ele_forward_medium OR jog_ele_backwards_medium THEN
    eleJogVelocity := joystick_velocity_medium;
ELSIF jog_ele_forward_slow OR jog_ele_backwards_slow THEN
    eleJogVelocity := joystick_velocity_slow;
END_IF

eleJogForwardTrig(CLK := eleJogForward);
eleJogBackwardsTrig(CLK := eleJogBackwards);

IF joystick_hold THEN
    ref.parts.ele.parts.virtualAxis.jog(eleJogForward, eleJogBackwards, eleJogVelocity, 0.0, 0.0);
ELSIF eleJogForwardTrig.Q THEN
    ref.parts.ele.processes.moveVelocity.request(units := AxesMoveVelocityUnits.DEGREES_PER_SECOND, eleJogVelocity);
ELSIF eleJogBackwardsTrig.Q THEN
    ref.parts.ele.processes.moveVelocity.request(units := AxesMoveVelocityUnits.DEGREES_PER_SECOND, -eleJogVelocity);
END_IF

joystick_disabled := jog_azi_disabled AND jog_ele_disabled;

END_FUNCTION_BLOCK

// ---- MTCS/Axes/Widgets/AxesManualJoystickRotWidget.TcPOU
FUNCTION_BLOCK AxesManualJoystickRotWidget
VAR_INPUT

    joystick_hold : BOOL := TRUE; 

    joystick_velocity_fast : LREAL := 6.0;   // degrees/s
    joystick_velocity_medium : LREAL := 1.0; // degrees/s
    joystick_velocity_slow : LREAL := 0.1;   // degrees/s
    
    jog_roc_forward_fast    : BOOL;
    jog_roc_forward_medium  : BOOL;
    jog_roc_forward_slow    : BOOL;
    jog_roc_backwards_fast    : BOOL;
    jog_roc_backwards_medium  : BOOL;
    jog_roc_backwards_slow    : BOOL;
    
    jog_ron_forward_fast    : BOOL;
    jog_ron_forward_medium  : BOOL;
    jog_ron_forward_slow    : BOOL;
    jog_ron_backwards_fast    : BOOL;
    jog_ron_backwards_medium  : BOOL;
    jog_ron_backwards_slow    : BOOL;
END_VAR
VAR_OUTPUT
    jog_roc_disabled : BOOL;
    jog_ron_disabled : BOOL;
    
    joystick_disabled : BOOL;
    
 
END_VAR
VAR_IN_OUT
    ref : Axes;
END_VAR
VAR
    rocJogForward : BOOL;
    rocJogBackwards : BOOL;
    rocJogVelocity : LREAL;
    ronJogForward : BOOL;
    ronJogBackwards : BOOL;
    ronJogVelocity : LREAL;
    
    rocJogForwardTrig : R_TRIG;
    rocJogBackwardsTrig : R_TRIG;
    ronJogForwardTrig : R_TRIG;
    ronJogBackwardsTrig : R_TRIG;
    
END_VAR

// rocmuth
IF joystick_hold THEN
    jog_roc_disabled := (NOT ref.parts.roc.parts.virtualAxis.isJogEnabled) OR ref.parts.roc.statuses.poweredStatus.disabled;
ELSE
    jog_roc_disabled := ref.parts.roc.processes.moveVelocity.statuses.enabledStatus.disabled OR ref.parts.roc.statuses.poweredStatus.disabled;
END_IF

rocJogForward   := jog_roc_forward_fast OR jog_roc_forward_medium OR jog_roc_forward_slow;
rocJogBackwards := jog_roc_backwards_fast OR jog_roc_backwards_medium OR jog_roc_backwards_slow;
IF jog_roc_forward_fast OR jog_roc_backwards_fast THEN
    rocJogVelocity := joystick_velocity_fast;
ELSIF jog_roc_forward_medium OR jog_roc_backwards_medium THEN
    rocJogVelocity := joystick_velocity_medium;
ELSIF jog_roc_forward_slow OR jog_roc_backwards_slow THEN
    rocJogVelocity := joystick_velocity_slow;
END_IF

rocJogForwardTrig(CLK := rocJogForward);
rocJogBackwardsTrig(CLK := rocJogBackwards);

IF joystick_hold THEN
    ref.parts.roc.parts.virtualAxis.jog(rocJogForward, rocJogBackwards, rocJogVelocity, 0.0, 0.0);
ELSIF rocJogForwardTrig.Q THEN
    ref.parts.roc.processes.moveVelocity.request(units := AxesMoveVelocityUnits.DEGREES_PER_SECOND, rocJogVelocity);
ELSIF rocJogBackwardsTrig.Q THEN
    ref.parts.roc.processes.moveVelocity.request(units := AxesMoveVelocityUnits.DEGREES_PER_SECOND, -rocJogVelocity);
END_IF

// ronvation
IF joystick_hold THEN
    jog_ron_disabled := (NOT ref.parts.ron.parts.virtualAxis.isJogEnabled) OR ref.parts.ron.statuses.poweredStatus.disabled;
ELSE
    jog_ron_disabled := ref.parts.ron.processes.moveVelocity.statuses.enabledStatus.disabled OR ref.parts.ron.statuses.poweredStatus.disabled;
END_IF

ronJogForward   := jog_ron_forward_fast OR jog_ron_forward_medium OR jog_ron_forward_slow;
ronJogBackwards := jog_ron_backwards_fast OR jog_ron_backwards_medium OR jog_ron_backwards_slow;
IF jog_ron_forward_fast OR jog_ron_backwards_fast THEN
    ronJogVelocity := joystick_velocity_fast;
ELSIF jog_ron_forward_medium OR jog_ron_backwards_medium THEN
    ronJogVelocity := joystick_velocity_medium;
ELSIF jog_ron_forward_slow OR jog_ron_backwards_slow THEN
    ronJogVelocity := joystick_velocity_slow;
END_IF

ronJogForwardTrig(CLK := ronJogForward);
ronJogBackwardsTrig(CLK := ronJogBackwards);

IF joystick_hold THEN
    ref.parts.ron.parts.virtualAxis.jog(ronJogForward, ronJogBackwards, ronJogVelocity, 0.0, 0.0);
ELSIF ronJogForwardTrig.Q THEN
    ref.parts.ron.processes.moveVelocity.request(units := AxesMoveVelocityUnits.DEGREES_PER_SECOND, ronJogVelocity);
ELSIF ronJogBackwardsTrig.Q THEN
    ref.parts.ron.processes.moveVelocity.request(units := AxesMoveVelocityUnits.DEGREES_PER_SECOND, -ronJogVelocity);
END_IF

joystick_disabled := jog_roc_disabled AND jog_ron_disabled;

END_FUNCTION_BLOCK

// ---- MTCS/Axes/Widgets/AxesManualOffsetsWidget.TcPOU
FUNCTION_BLOCK AxesManualOffsetsWidget
VAR_INPUT
    moveRelative : AxesMultiMoveProcessWIdget;
    pointRelative : AxesPointRelativeProcessWidget;
    alphaOffsetted : AxesAlphaWidget;
    deltaOffsetted : AxesDeltaWidget;
    rocTargetOffset : AxesAngleWidget;
    ronTargetOffset : AxesAngleWidget;
    aziTargetOffset : AxesAngleWidget;
    eleTargetOffset : AxesAngleWidget;
    preferMostTravel : BOOL;
END_VAR
VAR_OUTPUT
END_VAR
VAR_IN_OUT
    ref : Axes;
END_VAR
VAR
END_VAR



moveRelative(
    aziDisabled := ref.processes.moveRelative.statuses.enabledStatus.disabled OR ref.parts.azi.statuses.poweredStatus.disabled,
    eleDisabled := ref.processes.moveRelative.statuses.enabledStatus.disabled OR ref.parts.ele.statuses.poweredStatus.disabled,
    rocDisabled := ref.processes.moveRelative.statuses.enabledStatus.disabled OR ref.parts.roc.statuses.poweredStatus.disabled,
    ronDisabled := ref.processes.moveRelative.statuses.enabledStatus.disabled OR ref.parts.ron.statuses.poweredStatus.disabled,
    process := ref.processes.moveRelative,  
    title := 'Move relative');

pointRelative(
    alphaDisabled := ref.processes.pointRelative.statuses.enabledStatus.disabled OR ref.parts.azi.statuses.poweredStatus.disabled OR ref.parts.ele.statuses.poweredStatus.disabled,
    deltaDisabled := ref.processes.pointRelative.statuses.enabledStatus.disabled OR ref.parts.azi.statuses.poweredStatus.disabled OR ref.parts.ele.statuses.poweredStatus.disabled,
    rocDisabled := ref.processes.pointRelative.statuses.enabledStatus.disabled OR ref.parts.roc.statuses.poweredStatus.disabled,
    ronDisabled := ref.processes.pointRelative.statuses.enabledStatus.disabled OR ref.parts.ron.statuses.poweredStatus.disabled,
    units := moveRelative.units, // use the same units
    process := ref.processes.pointRelative,  
    title := 'Point relative');

alphaOffsetted(radians := ref.target.alphaOffsetted.radians.value);
deltaOffsetted(radians := ref.target.deltaOffsetted.radians.value);

aziTargetOffset(degrees := ref.parts.azi.targetOffset.degrees.value);
eleTargetOffset(degrees := ref.parts.ele.targetOffset.degrees.value);
rocTargetOffset(degrees := ref.parts.roc.targetOffset.degrees.value);
ronTargetOffset(degrees := ref.parts.ron.targetOffset.degrees.value);

END_FUNCTION_BLOCK

// ---- MTCS/Axes/Widgets/AxesMultiMoveProcessWidget.TcPOU
FUNCTION_BLOCK AxesMultiMoveProcessWidget
VAR_INPUT
    title : STRING;
    units : AxesMoveProcessWidgetUnits;
    
    actualStatus : StatusWidget;
    
    
    field_azi_sign : AxesDialogSign;
    field_azi_d : LREAL;
    field_azi_m : LREAL;
    field_azi_s : LREAL;
    field_azi_decimal : LREAL;
    
    field_ele_sign : AxesDialogSign;
    field_ele_d : LREAL;
    field_ele_m : LREAL;
    field_ele_s : LREAL;
    field_ele_decimal : LREAL;
    
    field_roc_sign : AxesDialogSign;
    field_roc_d : LREAL;
    field_roc_m : LREAL;
    field_roc_s : LREAL;
    field_roc_decimal : LREAL;
    
    field_ron_sign : AxesDialogSign;
    field_ron_d : LREAL;
    field_ron_m : LREAL;
    field_ron_s : LREAL;
    field_ron_decimal : LREAL;
    
    aziDisabled : BOOL;
    eleDisabled : BOOL;
    rocDisabled : BOOL;
    ronDisabled : BOOL;
    
    selected_azi : BOOL;
    selected_roc : BOOL;
    selected_ron : BOOL;
    selected_ele : BOOL;
END_VAR
VAR_OUTPUT
    unitsText : STRING;
    aziDeg : LREAL;
    eleDeg : LREAL;
    rocDeg : LREAL;
    ronDeg : LREAL;
    
    
END_VAR
VAR_IN_OUT
    process : AxesMultiMoveProcess;
END_VAR
VAR
END_VAR


actualStatus(
    text  := process.actualStatus,
    color := HealthBusyToColor(healthStatus := process.statuses.healthStatus, 
                               busyStatus   := process.statuses.busyStatus));

